// TIA Portal V17 program export: 17 tag tables, 178 data types, 56 data blocks, 100 code blocks (in call order from the OBs), 30 instance data blocks

VAR_GLOBAL   // PLC tag table "Default tag table"
   TIMER_PF_FEEDER_1_UNIT_01_LINE_1 AT %T21 : Timer;
   TIMER_PF_FEEDER_1_UNIT_01_LINE_2 AT %T22 : Timer;
   TIMER_PF_FEEDER_1_UNIT_02_LINE_1 AT %T23 : Timer;
   TIMER_PF_FEEDER_1_UNIT_02_LINE_2 AT %T24 : Timer;
   "Clock_Byte(1)" AT %MB0 : Byte;
   OK_DEL_NCU AT %M710.0 : Bool;
   Tag_1 AT %M45.0 : Bool;
   Tag_2 AT %M250.0 : Bool;
   Tag_3 AT %M71.0 : Bool;
   Tag_4 AT %M71.1 : Bool;
   Tag_5 AT %M71.2 : Bool;
   Tag_6 AT %M71.3 : Bool;
   Tag_7 AT %M71.4 : Bool;
   U01_OERLIKON_1_LINE_1_MEDICOAT_TIMER AT %T39 : Timer;   // UNIT 01 OERLIKON 1 LINE 1 MEDICOAT TIMER
   U01_OERLIKON_1_LINE_2_MEDICOAT_TIMER AT %T40 : Timer;   // UNIT 01 OERLIKON 1 LINE 2 MEDICOAT TIMER
   U02_OERLIKON_1_LINE_1_MEDICOAT_TIMER AT %T41 : Timer;   // UNIT 02 OERLIKON 1 LINE 1 MEDICOAT TIMER
   U02_OERLIKON_1_LINE_2_MEDICOAT_TIMER AT %T42 : Timer;   // UNIT 02 OERLIKON 1 LINE 2 MEDICOAT TIMER
   U01_COMBINER_MEDICOAT_TIMER AT %T44 : Timer;   // UNIT 01 COMBINER MEDICOAT TIMER
   U02_COMBINER_MEDICOAT_TIMER AT %T45 : Timer;   // UNIT 02 COMBINER MEDICOAT TIMER
   U01_LASER_HEAD_MEDICOAT_TIMER AT %T46 : Timer;   // UNIT 01 LASER HEAD MEDICOAT TIMER
   U02_LASER_HEAD_MEDICOAT_TIMER AT %T47 : Timer;   // UNIT 02 LASER HEAD MEDICOAT TIMER
   UNIT_01_PF1_L2_PRESS AT %MD26 : Real;
   UNIT_01_PF1_L1_PRESS AT %MD30 : Real;
   UNIT_01_PF2_L1_PRESS AT %MD34 : Real;
   U02_OERLIKON_2_LINE_2_MEDICOAT_TIMER AT %T43 : Timer;   // UNIT 02 OERLIKON 2 LINE 1 MEDICOAT TIMER
   TIMER_PF_FEEDER_2_UNIT_02_LINE_2 AT %T25 : Timer;
   Tag_8 AT %M445.4 : Bool;
   Tag_9 AT %T26 : Timer;
   Tag_10 AT %IW1810 : Int;
   COUNT_ANDER AT %MW448 : Int;
   PB_HOPPERS_MANUAL_MODE_SELECTED_LIGHT_Q AT %Q141.4 : Bool;   // MANUAL MODE SELECTED LIGHT OUTPUT
END_VAR

VAR_GLOBAL   // PLC tag table "TAGS_MARKS"
   Clock_Byte AT %MB1 : Byte;
   "M_0.1_SEC_10HZ" AT %M1.0 : Bool;   // 10HZ 0.1SEC
   "M_0.2_SEC_5Hz" AT %M1.1 : Bool;   // 5HZ 0.2SEC
   "M_0.4_SEC_2.5HZ" AT %M1.2 : Bool;   // 2.5HZ 0.4SEC
   "M_0.5_SEC_2HZ" AT %M1.3 : Bool;   // 2HZ 0.5SEC
   "M_0.8_SEC_1.25HZ" AT %M1.4 : Bool;   // 2.25HZ 0.8SEC
   "M_1.6_SEC_625HZ" AT %M1.6 : Bool;   // 0.625HZ 1.6SEC
   M_1_SEC_1HZ AT %M1.5 : Bool;   // 1HZ 1.0SEC
   "M_2_SEC_0.5HZ" AT %M1.7 : Bool;   // 0.5HZ 2.0SEC
   M_DUMMY_OFF AT %M0.3 : Bool;   // DUMMY OFF
   M_DUMMY_ON AT %M0.2 : Bool;   // DUMMY ON
   M_DUMMY_OUT AT %M0.4 : Bool;   // DUMMY OUT
   M_FIRST_SCAN AT %M0.6 : Bool;   // M FIRST SCAN
   M_NEW_START AT %M0.5 : Bool;   // NEW START / M NEW START
   M_ONE AT %M0.1 : Bool;   // ALWAYS ON
   M_REVISAR_FALTA_ALGO AT %M2.3 : Bool;   // REVISAR FALTA ALGO DE PROGRAMACIÓN
   M_TEMPORARY_USE_OEM AT %M5.0 : Bool;   // M_TEMPORARY_USE_OEM(CONFIGURE CORRECTLY AND DELETE) / M FOR TEMPORARY USE (OEM)
   M_ZERO AT %M0.0 : Bool;   // ALWAYS OFF
   NETWORK_CHECK AT %M0.7 : Bool;   // ADAPT NETWORK LOGIC ACCORDING TO MACHINE STRUCTURE
   Softkey_Input_Byte AT %IB124 : Byte;
END_VAR

VAR_GLOBAL   // PLC tag table "TAGS_IO_MPP_ITC_IPC_HT10"
   HT10_INS AT %I0.0 : "HT10_INPUTS";   // HT10 INPUTS
   HT10_OUTS AT %Q0.0 : "HT10_OUTPUTS";   // HT10 OUTPUTS
   MPP_INS AT %I120.0 : "MPP_INPUTS";   // MPP INPUTS
   MPP_OUT AT %Q120.0 : "MPP_OUTPUTS";   // MPP OUTPUTS
   TOUCH_PANEL_INPUT_1 AT %IB138 : Byte;   // TOUCH PANEL INPUT BYTE 1
   TOUCH_PANEL_INPUT_2 AT %IB139 : Byte;   // TOUCH PANEL INPUT BYTE 2
END_VAR

VAR_GLOBAL   // PLC tag table "TEMPORAL_TAG_PANI"
   PART_PRESENT_SENSOR_UNIT_1 AT %MW5000 : Int;
   Delay_Z11_Start AT %T10 : Timer;
   Delay_Z21_Start AT %T20 : Timer;
   U01_STA4_BRUSH_WORN_ALARM AT %M100.0 : Bool;
   U01_STA4_BRUSH_WORN_INPUT AT %M100.1 : Bool;
   U01_STA4_BRUSH_CHANGE_ACK AT %M100.2 : Bool;
END_VAR

VAR_GLOBAL   // PLC tag table "TAGS_IO_GENERAL_CLADDING"
   "/////_CRM_/////" AT %M6060.0 : Bool;   // /////_CRM_/////
   "/////_ELECTRICAL_CABINET_/////" AT %M6100.0 : Bool;   // /////_ELECTRICAL_CABINET_/////
   "/////_LINE_CONTACTOR_/////" AT %M6200.0 : Bool;   // /////_LINE_CONTACTOR_/////
   "/////_MPP_AND_SIGNAL_TOWER_/////" AT %M141.0 : Bool;   // /////_MPP_AND_SIGNAL_TOWER_/////
   "/////_POWER_SUPPLY_/////" AT %M6080.0 : Bool;   // /////_POWER_SUPPLY_/////
   "/////_SAFETY_DOORS_/////" AT %M6180.0 : Bool;   // /////_SAFETY_DOORS_/////
   CIRCUIT_BREAKER_230VAC_TRIPPED AT %I140.1 : Bool;   // 230 VAC CIRCUIT BREAKER TRIPPED
   CIRCUIT_BREAKER_FC04_TRIPPED AT %I140.0 : Bool;   // FC04 CIRCUIT BREAKER TRIPPED. FAN.
   CIRCUIT_BREAKER_FC35_1_TRIPPED AT %I140.5 : Bool;   // FC35.1 CIRCUIT BREAKER TRIPPED
   CIRCUIT_BREAKER_FC35_2_TRIPPED AT %I140.6 : Bool;   // FC35.2 CIRCUIT BREAKER TRIPPED
   CIRCUIT_BREAKER_FC35_3_TRIPPED AT %I140.7 : Bool;   // FC35.3 CIRCUIT BREAKER TRIPPED
   CONTROL_ON_Q AT %Q140.0 : Bool;   // CONTROL ON OUTPUT
   MAIN_CIRCUIT_BREAKER_I AT %M580.1 : Bool;   // MAIN CABINET CIRCUIT BREAKER TRIPPED INPUT
   PB_AUTO_CYCLE_LIGHT_Q AT %Q141.1 : Bool;   // AUTOMATIC CYCLE LIGHT OUTPUT
   PB_AUTO_MODE_SELECTED_LIGHT_Q AT %Q141.2 : Bool;   // AUTOMATIC MODE SELECTED LIGHT OUTPUT
   PB_IMMEDIATE_STOP_I AT %I144.3 : Bool;   // IMMEDIATE STOP INPUT
   PB_MANUAL_MODE_SELECTED_LIGHT_Q AT %Q141.3 : Bool;   // MANUAL MODE SELECTED LIGHT OUTPUT
   PB_RESET_FAULTS_I AT %I144.6 : Bool;   // RESET FAULTS INPUT
   PB_START_CYCLE_I AT %I144.2 : Bool;   // START CYCLE INPUT
   PS_24V_NOT_READY_DEV_1_I AT %I142.2 : Bool;   // POWER SUPPLY 24V NOT READY DEVICE 1 INPUT
   PS_24V_NOT_READY_DEV_2_I AT %I142.3 : Bool;   // POWER SUPPLY 24V NOT READY DEVICE 2 INPUT
   SIGNAL_TWR_BLUE_LIGHT_Q AT %M141.1 : Bool;   // SIGNAL TOWER BLUE LIGHT OUTPUT
   SIGNAL_TWR_GREEN_LIGHT_Q AT %Q141.5 : Bool;   // SIGNAL TOWER GREEN LIGHT OUTPUT
   SIGNAL_TWR_HOOTER_Q AT %M141.3 : Bool;   // SIGNAL TOWER HOOTER LIGHT OUTPUT
   SIGNAL_TWR_RED_LIGHT_Q AT %Q141.7 : Bool;   // SIGNAL TOWER RED LIGHT OUTPUT
   SIGNAL_TWR_WHITE_LIGHT_Q AT %M141.2 : Bool;   // SIGNAL TOWER WHITE LIGHT OUTPUT
   SIGNAL_TWR_YELLOW_LIGHT_Q AT %Q141.6 : Bool;   // SIGNAL TOWER YELLOW LIGHT OUTPUT
   PB_HOPPERS_AUTO_MODE_SELECTED_LIGHT_Q AT %Q141.0 : Bool;   // AUTOMATIC MODE SELECTED LIGHT OUTPUT
   PB_FEEDERS_AUTOMATIC_MODE_SELECT_I AT %I144.0 : Bool;   // AUTOMATIC MODE SELECT INPUT
   PB_FEEDERS_MANUAL_MODE_SELECT_I AT %I144.1 : Bool;   // MANUAL MODE SELECT INPUT
   PB_HOPPERS_MANUAL_MODE_SELECT_I AT %I142.6 : Bool;   // MANUAL MODE SELECT INPUT
   PB_HOPPERS_AUTOMATIC_MODE_SELECT_I AT %I142.5 : Bool;   // AUTOMATIC MODE SELECT INPUT
END_VAR

VAR_GLOBAL   // PLC tag table "TAGS_IO_HOPPERS_CLADDING"
   "//////////_HOPPERS_POWDER_FLOW_SENSORS_//////////" AT %M580.0 : Bool;
   "//////////_HOPPERS_WEIGHT_CONTROL_SENSORS_//////////" AT %M596.0 : Bool;
   "/////_HOPPER_JACKET_TEMPERATURE_CONTROL_/////" AT %M150.0 : Bool;   // /////_HOPPER_JACKET_TEMPERATURE_CONTROL/////
   "/////_HOPPER_LEVEL_SENSORS_/////" AT %M70.0 : Bool;   // /////_HOPPER_LEVEL_SENSORS_/////
   "/////_HOPPER_PRESSURE_SENSORS/////" AT %M510.0 : Bool;   // /////_HOPPER_PRESSURE_SENSORS/////
   "/////_HOPPERS_PRESSURE_CONTROLS_/////" AT %M160.0 : Bool;
   "/////_HOPPERS_VALVES_/////" AT %M75.0 : Bool;   // /////_HOPPERS_VALVES_/////
   HPPR_1_MOTOR_ENABLE_1 AT %Q140.4 : Bool;   // HOPPER 1 MOTOR ENABLE SIGNAL 1
   HPPR_1_MOTOR_ENABLE_2 AT %Q140.5 : Bool;   // HOPPER 1 MOTOR ENABLE SIGNAL 2
   HPPR_2_MOTOR_ENABLE_1 AT %Q140.6 : Bool;   // HOPPER 2 MOTOR ENABLE SIGNAL 1
   HPPR_2_MOTOR_ENABLE_2 AT %Q140.7 : Bool;   // HOPPER 2 MOTOR ENABLE SIGNAL 2
   HPPR_3_MOTOR_ENABLE_1 AT %Q142.2 : Bool;   // HOPPER 3 MOTOR ENABLE SIGNAL 1
   HPPR_3_MOTOR_ENABLE_2 AT %Q142.3 : Bool;   // HOPPER 3 MOTOR ENABLE SIGNAL 2
   HPPR_4_MOTOR_ENABLE_1 AT %Q142.4 : Bool;   // HOPPER 4 MOTOR ENABLE SIGNAL 1
   HPPR_4_MOTOR_ENABLE_2 AT %Q142.5 : Bool;   // HOPPER 4 MOTOR ENABLE SIGNAL 2
   HPPR_5_MOTOR_ENABLE_1 AT %Q142.6 : Bool;   // HOPPER 5 MOTOR ENABLE SIGNAL 1
   HPPR_5_MOTOR_ENABLE_2 AT %Q142.7 : Bool;   // HOPPER 5 MOTOR ENABLE SIGNAL 2
   U01_HOPPER_1_HIGH_LEVEL_SENSOR_I AT %I70.1 : Bool;   // UNIT 01 HOPPER 1 HIGH LEVEL SENSOR INPUT
   U01_HOPPER_1_LOW_LEVEL_SENSOR_I AT %I70.0 : Bool;   // UNIT 01 HOPPER 1 LOW LEVEL SENSOR INPUT
   U01_HOPPER_1_LOWER_JACKET_TEMP_CONTROL_I AT %MW162 : Word;   // UNIT 01 HOPPER 1 LOWER JACKET TEMPERATURE CONTROL INPUT
   U01_HOPPER_1_LOWER_JACKET_TEMP_CONTROL_Q AT %MW166 : Word;   // UNIT 01 HOPPER 1 LOWER JACKET TEMPERATURE CONTROL OUTPUT
   U01_HOPPER_1_POWDER_FLOW_SENSOR_I AT %IW580 : Word;   // UNIT 01 HOPPER 1 POWDER FLOW SENSOR INPUT
   U01_HOPPER_1_PRESSURE_SENSOR_I AT %IW510 : Word;   // UNIT 01HOPPER 1 PRESSURE SENSOR INPUT
   U01_HOPPER_1_UPPER_JACKET_TEMP_CONTROL_I AT %MW150 : Word;   // UNIT 01 HOPPER 1 UPPER JACKET TEMPERATURE CONTROL INPUT
   U01_HOPPER_1_UPPER_JACKET_TEMP_CONTROL_Q AT %MW155 : Word;   // UNIT 01 HOPPER 1 UPPER JACKET TEMPERATURE CONTROL OUTPUT
   U01_HOPPER_1_WEIGHT_SENSOR_I AT %IW596 : Word;   // UNIT 01 HOPPER 1 WEIGHT SENSOR INPUT
   U01_HOPPER_2_HIGH_LEVEL_SENSOR_I AT %I70.3 : Bool;   // UNIT 01 HOPPER 2 HIGH LEVEL SENSOR INPUT
   U01_HOPPER_2_LOW_LEVEL_SENSOR_I AT %I70.2 : Bool;   // UNIT 01 HOPPER 2 LOW LEVEL SENSOR INPUT
   U01_HOPPER_2_LOWER_JACKET_TEMP_CONTROL_I AT %MW168 : Word;   // UNIT 01 HOPPER 2 LOWER JACKET TEMPERATURE CONTROL INPUT
   U01_HOPPER_2_LOWER_JACKET_TEMP_CONTROL_Q AT %MW172 : Word;   // UNIT 01 HOPPER 2 LOWER JACKET TEMPERATURE CONTROL OUTPUT
   U01_HOPPER_2_POWDER_FLOW_SENSOR_I AT %IW582 : Word;   // UNIT 01 HOPPER 2 POWDER FLOW SENSOR INPUT
   U01_HOPPER_2_PRESSURE_SENSOR_I AT %IW518 : Word;   // UNIT 01HOPPER 2 PRESSURE SENSOR INPUT
   U01_HOPPER_2_UPPER_JACKET_TEMP_CONTROL_I AT %MW151 : Word;   // UNIT 01 HOPPER 2 UPPER JACKET TEMPERATURE CONTROL INPUT
   U01_HOPPER_2_UPPER_JACKET_TEMP_CONTROL_Q AT %MW156 : Word;   // UNIT 01 HOPPER 2 UPPER JACKET TEMPERATURE CONTROL OUTPUT
   U01_HOPPER_2_WEIGHT_SENSOR_I AT %IW598 : Word;   // UNIT 01 HOPPER 2 WEIGHT SENSOR INPUT
   U01_HPPR_1_CLEANING_VALVE_Q AT %M73.5 : Bool;   // UNIT 01 HOPPER 1 CLEANING VALVE OUTPUT
   U01_HPPR_1_FEEDBACK_PRESSURE_CONTROL_I AT %IW160 : Int;   // UNIT 01 HOPPER 1 FEEDBACK PRESSURE CONTROL INPUT
   U01_HPPR_1_PRESSURE_CONTROL_Q AT %QW160 : Int;   // UNIT 01 HOPPER 1 PRESSURE CONTROL OUTPUT
   U01_HPPR_1_PRESSURIZE_GAS_VALVE_Q AT %Q70.0 : Bool;   // UNIT 01 HOPPER 1 PRESSURIZE GAS VALVE OUTPUT
   U01_HPPR_1_RELIEF_GAS_VALVE_Q AT %Q70.1 : Bool;   // UNIT 01 HOPPER 1 RELIEF GAS VALVE OUTPUT
   U01_HPPR_1_TRANSF_POWDER_VALVE_Q AT %M1500.0 : Bool;   // UNIT 01 HOPPER 1 TRANSFER POWDER VALVE OUTPUT
   U01_HPPR_2_CLEANING_VALVE_Q AT %M73.6 : Bool;   // UNIT 01 HOPPER 2 CLEANING VALVE OUTPUT
   U01_HPPR_2_FEEDBACK_PRESSURE_CONTROL_I AT %IW162 : Int;   // UNIT 01 HOPPER 2 FEEDBACK PRESSURE CONTROL INPUT
   U01_HPPR_2_PRESSURE_CONTROL_Q AT %QW162 : Int;   // UNIT 01 HOPPER 2 PRESSURE CONTROL OUTPUT
   U01_HPPR_2_PRESSURIZE_GAS_VALVE_Q AT %Q70.2 : Bool;   // UNIT 01 HOPPER 2 PRESSURIZE GAS VALVE OUTPUT
   U01_HPPR_2_RELIEF_GAS_VALVE_Q AT %Q70.3 : Bool;   // UNIT 01 HOPPER 2 RELIEF GAS VALVE OUTPUT
   U01_HPPR_2_TRANSF_POWDER_VALVE_Q AT %M1500.1 : Bool;   // UNIT 01 HOPPER 2 TRANSFER POWDER VALVE OUTPUT
   U02_HOPPER_1_HIGH_LEVEL_SENSOR_I AT %I70.5 : Bool;   // UNIT 02 HOPPER 1 HIGH LEVEL SENSOR INPUT
   U02_HOPPER_1_LOW_LEVEL_SENSOR_I AT %I70.4 : Bool;   // UNIT 02 HOPPER 1 LOW LEVEL SENSOR INPUT
   U02_HOPPER_1_LOWER_JACKET_TEMP_CONTROL_I AT %MW176 : Word;   // UNIT 02 HOPPER 1 LOWER JACKET TEMPERATURE CONTROL INPUT
   U02_HOPPER_1_LOWER_JACKET_TEMP_CONTROL_Q AT %MW178 : Word;   // UNIT 02 HOPPER 1 LOWER JACKET TEMPERATURE CONTROL OUTPUT
   U02_HOPPER_1_POWDER_FLOW_SENSOR_I AT %IW584 : Word;   // UNIT 02 HOPPER 1 POWDER FLOW SENSOR INPUT
   U02_HOPPER_1_PRESSURE_SENSOR_I AT %IW526 : Word;   // UNIT 02 HOPPER 1 PRESSURE SENSOR INPUT
   U02_HOPPER_1_UPPER_JACKET_TEMP_CONTROL_I AT %MW152 : Word;   // UNIT 02 HOPPER 1 UPPER JACKET TEMPERATURE CONTROL INPUT
   U02_HOPPER_1_UPPER_JACKET_TEMP_CONTROL_Q AT %MW157 : Word;   // UNIT 02 HOPPER 1 UPPER JACKET TEMPERATURE CONTROL OUTPUT
   U02_HOPPER_1_WEIGHT_SENSOR_I AT %IW600 : Word;   // UNIT 02 HOPPER 1 WEIGHT SENSOR INPUT
   U02_HOPPER_2_HIGH_LEVEL_SENSOR_I AT %I70.7 : Bool;   // UNIT 02 HOPPER 2 HIGH LEVEL SENSOR INPUT
   U02_HOPPER_2_LOW_LEVEL_SENSOR_I AT %I70.6 : Bool;   // UNIT 02 HOPPER 2 LOW LEVEL SENSOR INPUT
   U02_HOPPER_2_LOWER_JACKET_TEMP_CONTROL_I AT %MW164 : Word;   // UNIT 02 HOPPER 2 LOWER JACKET TEMPERATURE CONTROL INPUT
   U02_HOPPER_2_LOWER_JACKET_TEMP_CONTROL_Q AT %MW174 : Word;   // UNIT 02 HOPPER 2 LOWER JACKET TEMPERATURE CONTROL OUTPUT
   U02_HOPPER_2_POWDER_FLOW_SENSOR_I AT %IW588 : Word;   // UNIT 02 HOPPER 2 POWDER FLOW SENSOR INPUT
   U02_HOPPER_2_PRESSURE_SENSOR_I AT %IW534 : Word;   // UNIT 02 HOPPER 2 PRESSURE SENSOR INPUT
   U02_HOPPER_2_UPPER_JACKET_TEMP_CONTROL_I AT %MW153 : Word;   // UNIT 02 HOPPER 2 UPPER JACKET TEMPERATURE CONTROL INPUT
   U02_HOPPER_2_UPPER_JACKET_TEMP_CONTROL_Q AT %MW158 : Word;   // UNIT 02 HOPPER 2 UPPER JACKET TEMPERATURE CONTROL OUTPUT
   U02_HOPPER_2_WEIGHT_SENSOR_I AT %IW602 : Word;   // UNIT 02 HOPPER 2 WEIGHT SENSOR INPUT
   U02_HOPPER_3_HIGH_LEVEL_SENSOR_I AT %I71.1 : Bool;   // UNIT 02 HOPPER 3 HIGH LEVEL SENSOR INPUT
   U02_HOPPER_3_LOW_LEVEL_SENSOR_I AT %I71.0 : Bool;   // UNIT 02 HOPPER 3 LOW LEVEL SENSOR INPUT
   U02_HOPPER_3_LOWER_JACKET_TEMP_CONTROL_I AT %MW170 : Word;   // UNIT 02 HOPPER 3 LOWER JACKET TEMPERATURE CONTROL INPUT
   U02_HOPPER_3_LOWER_JACKET_TEMP_CONTROL_Q AT %MW180 : Word;   // UNIT 02 HOPPER 3 LOWER JACKET TEMPERATURE CONTROL OUTPUT
   U02_HOPPER_3_POWDER_FLOW_SENSOR_I AT %IW590 : Word;   // UNIT 02 HOPPER 3 POWDER FLOW SENSOR INPUT
   U02_HOPPER_3_PRESSURE_SENSOR_I AT %IW542 : Word;   // UNIT 02 HOPPER 3 PRESSURE SENSOR INPUT
   U02_HOPPER_3_UPPER_JACKET_TEMP_CONTROL_I AT %MW154 : Word;   // UNIT 02 HOPPER 3 UPPER JACKET TEMPERATURE CONTROL INPUT
   U02_HOPPER_3_UPPER_JACKET_TEMP_CONTROL_Q AT %MW159 : Word;   // UNIT 02 HOPPER 3 UPPER JACKET TEMPERATURE CONTROL OUTPUT
   U02_HOPPER_3_WEIGHT_SENSOR_I AT %IW586 : Word;   // UNIT 02 HOPPER 3 WEIGHT SENSOR INPUT
   U02_HPPR_1_CLEANING_VALVE_Q AT %M73.7 : Bool;   // UNIT 02 HOPPER 1 CLEANING VALVE OUTPUT
   U02_HPPR_1_FEEDBACK_PRESSURE_CONTROL_I AT %IW164 : Int;   // UNIT 02 HOPPER 1 FEEDBACK PRESSURE CONTROL INPUT
   U02_HPPR_1_PRESSURE_CONTROL_Q AT %QW164 : Int;   // UNIT 02 HOPPER 1 PRESSURE CONTROL OUTPUT
   U02_HPPR_1_PRESSURIZE_GAS_VALVE_Q AT %Q70.4 : Bool;   // UNIT 02 HOPPER 1 PRESSURIZE GAS VALVE OUTPUT
   U02_HPPR_1_RELIEF_GAS_VALVE_Q AT %Q70.5 : Bool;   // UNIT 02 HOPPER 1 RELIEF GAS VALVE OUTPUT
   U02_HPPR_1_TRANSF_POWDER_VALVE_Q AT %M1500.2 : Bool;   // UNIT 02 HOPPER 1 TRANSFER POWDER VALVE OUTPUT
   U02_HPPR_2_CLEANING_VALVE_Q AT %M74.0 : Bool;   // UNIT 02 HOPPER 2 CLEANING VALVE OUTPUT
   U02_HPPR_2_FEEDBACK_PRESSURE_CONTROL_I AT %IW166 : Int;   // UNIT 02 HOPPER 2 FEEDBACK PRESSURE CONTROL INPUT
   U02_HPPR_2_PRESSURE_CONTROL_Q AT %QW166 : Int;   // UNIT 02 HOPPER 2 PRESSURE CONTROL OUTPUT
   U02_HPPR_2_PRESSURIZE_GAS_VALVE_Q AT %Q70.6 : Bool;   // UNIT 02 HOPPER 2 PRESSURIZE GAS VALVE OUTPUT
   U02_HPPR_2_RELIEF_GAS_VALVE_Q AT %Q70.7 : Bool;   // UNIT 02 HOPPER 2 RELIEF GAS VALVE OUTPUT
   U02_HPPR_2_TRANSF_POWDER_VALVE_Q AT %M1500.3 : Bool;   // UNIT 02 HOPPER 2 TRANSFER POWDER VALVE OUTPUT
   U02_HPPR_3_CLEANING_VALVE_Q AT %M1500.5 : Bool;   // UNIT 02 HOPPER 3 CLEANING VALVE OUTPUT
   U02_HPPR_3_FEEDBACK_PRESSURE_CONTROL_I AT %IW168 : Int;   // UNIT 02 HOPPER 3 FEEDBACK PRESSURE CONTROL INPUT
   U02_HPPR_3_PRESSURE_CONTROL_Q AT %QW170 : Int;   // UNIT 02 HOPPER 3 PRESSURE CONTROL OUTPUT
   U02_HPPR_3_PRESSURIZE_GAS_VALVE_Q AT %Q71.0 : Bool;   // UNIT 02 HOPPER 3 PRESSURIZE GAS VALVE OUTPUT
   U02_HPPR_3_RELIEF_GAS_VALVE_Q AT %Q71.1 : Bool;   // UNIT 02 HOPPER 3 RELIEF GAS VALVE OUTPUT
   U02_HPPR_3_TRANSF_POWDER_VALVE_Q AT %M1500.4 : Bool;   // UNIT 02 HOPPER 3 TRANSFER POWDER VALVE OUTPUT
END_VAR

VAR_GLOBAL   // PLC tag table "TAGS_IO_POWDER_FEEDERS_CLADDING"
   "//////////PF_HOPPERS_PRESSURE_SENSORS//////////" AT %M810.0 : Bool;
   "//////////POWDER_FEEDER_WEIGHT_CONTROL//////////" AT %M712.0 : Bool;
   "//////////POWDER_FLOW_SENSORS//////////" AT %M700.0 : Bool;
   U01_PF_1_WEIGHT_SENSOR_I AT %IW712 : Word;   // UNIT 01 POWDER FEEDER 1 WEIGHT SENSOR INPUT
   U02_COMBINER_FLOW_SENSOR_I AT %IW1706 : Word;   // UNIT 02 COMBINER FLOW SENSOR INPUT
   U02_OERLIKON_2_LINE_2_MEDICOAT_FLOW_CONTROL AT %MW16 : UInt;   // UNIT 02 OERLIKON 2 LINE 2 MEDICOAT FLOW CONTROL
   U02_OERLIKON_1_LINE_1_MEDICOAT_FLOW_CONTROL AT %IW1700 : Int;   // UNIT 02 OERLIKON 1 LINE 1 MEDICOAT FLOW CONTROL
   U02_COMBINER_MEDICOAT_FLOW_CONTROL AT %IW1708 : Int;   // UNIT 02 COMBINER MEDICOAT FLOW CONTROL
   U02_OERLIKON_2_LINE_1_MEDICOAT_FLOW_CONTROL AT %IW1704 : Int;   // UNIT 02 OERLIKON 2 LINE 1 MEDICOAT FLOW CONTROL
   U01_OERLIKON_1_LINE_1_MEDICOAT_FLOW_CONTROL AT %IW700 : Int;   // UNIT 01 OERLIKON 1 LINE 1 MEDICOAT FLOW CONTROL
   U02_PF_1_HPPR_1_PRESSURE_SENSOR_I AT %IW1818 : Word;   // UNIT 02 POWDER FEEDER 1 HOPPER 1 PRESSURE SENSOR INPUT
   U01_PF_1_HPPR_1_FLOW_SENSOR_I AT %MW700 : Word;   // UNIT 01 POWDER FEEDER 1 HOPPER 1 FLOW SENSOR INPUT
   U02_PF_2_HPPR_1_FLOW_SENSOR_I AT %MW1704 : Word;   // UNIT 02 POWDER FEEDER 2 HOPPER 1 FLOW SENSOR INPUT
   U01_PF_1_HPPR_1_PRESSURE_SENSOR_I AT %IW810 : Word;   // UNIT 01 POWDER FEEDER 1 HOPPER 1 PRESSURE SENSOR INPUT
   U02_PF_1_WEIGHT_SENSOR_I AT %MW1712 : Word;   // UNIT 02 POWDER FEEDER 1 WEIGHT SENSOR INPUT
   U02_PF_2_HPPR_1_PRESSURE_SENSOR_I AT %IW1822 : Word;   // UNIT 02 POWDER FEEDER 2 HOPPER 1 PRESSURE SENSOR INPUT
   U02_LASER_HEAD_FLOW_SENSOR_I AT %MW1708 : Word;   // UNIT 02 LASER HEAD FLOW SENSOR INPUT
   U02_PF_1_HPPR_2_PRESSURE_SENSOR_I AT %IW1820 : Word;   // UNIT 02 POWDER FEEDER 1 HOPPER 2 PRESSURE SENSOR INPUT
   U01_PF_1_HPPR_2_PRESSURE_SENSOR_I AT %IW812 : Word;   // UNIT 01 POWDER FEEDER 1 HOPPER 2 PRESSURE SENSOR INPUT
   U02_OERLIKON_1_LINE_2_MEDICOAT_FLOW_CONTROL AT %IW1702 : Int;   // UNIT 02 OERLIKON 1 LINE 2 MEDICOAT FLOW CONTROL
   U01_LASER_HEAD_FLOW_SENSOR_I AT %MW706 : Word;   // UNIT 01 LASER HEAD FLOW SENSOR INPUT
   U02_PF_2_WEIGHT_SENSOR_I AT %MW1714 : Word;   // UNIT 02 POWDER FEEDER 2 WEIGHT SENSOR INPUT
   U01_COMBINER_MEDICOAT_FLOW_CONTROL AT %IW708 : Int;   // UNIT 01 COMBINER MEDICOAT FLOW CONTROL
   U02_LASER_HEAD_MEDICOAT_CONTROL AT %IW1710 : Int;   // UNIT 02 LASER HEAD MEDICOAT FLOW CONTROL
   U01_COMBINER_FLOW_SENSOR_I AT %MW704 : Word;   // UNIT 01 COMBINER FLOW SENSOR INPUT
   U02_PF_1_HPPR_2_FLOW_SENSOR_I AT %MW1702 : Word;   // UNIT 02 POWDER FEEDER 1 HOPPER 2 FLOW SENSOR INPUT
   U01_OERLIKON_1_LINE_2_MEDICOAT_FLOW_CONTROL AT %IW702 : Int;   // UNIT 01 OERLIKON 1 LINE 2 MEDICOAT FLOW CONTROL
   U01_PF_1_HPPR_2_FLOW_SENSOR_I AT %MW702 : Word;   // UNIT 01 POWDER FEEDER 1 HOPPER 2 FLOW SENSOR INPUT
   U02_PF_1_HPPR_1_FLOW_SENSOR_I AT %MW1700 : Word;   // UNIT 02 POWDER FEEDER 1 HOPPER 1 FLOW SENSOR INPUT
   U01_LASER_HEAD_MEDICOAT_CONTROL AT %IW710 : Int;   // UNIT 01 LASER HEAD MEDICOAT FLOW CONTROL
   U02_PF1_L2_STIRRER_CURRENT AT %IW1716 : Int;
   U02_PF1_L1_STIRRER_CURRENT AT %IW1712 : Int;
   U02_PF2_L1_DISK_CURRENT AT %IW1722 : Int;
   U02_PF1_L2_DISK_CURRENT AT %IW1718 : Int;
   U01_PF1_L2_DISK_CURRENT AT %IW722 : Int;
   U01_PF1_L1_DISK_CURRENT AT %IW718 : Int;
   U01_PF1_L2_STIRRER_CURRENT AT %IW720 : Int;
   U01_PF1_L1_STIRRER_CURRENT AT %IW716 : Int;
   U02_PF1_L1_DISK_CURRENT AT %IW1714 : Int;
   U02_PF2_L2_STIRRER_CURRENT AT %IW1720 : Int;
END_VAR

VAR_GLOBAL   // PLC tag table "TAGS_IO_SERVICES_CLADDING"
   "/////_COOLING_CHILLER_/////" AT %M8305.6 : Bool;   // /////_COOLING_CHILLER_/////
   "/////_OTHER_CIRCUIT_BREAKERS_/////" AT %M8308.0 : Bool;   // /////_OTHER_CIRCUIT_BREAKERS_/////
   "/////_OTHER_CONTACTOR_/////" AT %M8309.5 : Bool;   // /////_OTHER_CONTACTOR_/////
END_VAR

VAR_GLOBAL   // PLC tag table "TAGS_IO_STIRRERS_CLADDING"
   "//////////_STIRRER_UNIT_01_HOPPER_1_//////////" AT %M500.0 : Bool;
   "//////////_STIRRER_UNIT_01_HOPPER_2_//////////" AT %M600.0 : Bool;
   "//////////_STIRRER_UNIT_02_HOPPER_1_//////////" AT %M2000.0 : Bool;
   "//////////_STIRRER_UNIT_02_HOPPER_2_//////////" AT %M800.0 : Bool;
   "//////////_STIRRER_UNIT_02_HOPPER_3_//////////" AT %M900.0 : Bool;
   U01_HPPR_1_STRR_ACTUAL_PHASE_CURRENT_FILTERED_INPUT AT %ID3016 : DInt;   // UNIT 01 HOPPER 1 STIRRER ACTUAL PHASE CURRENT FILTERED INPUT
   U01_HPPR_1_STRR_ACTUAL_PHASE_CURRENT_INPUT AT %ID3012 : DInt;   // UNIT 01 HOPPER 1 STIRRER ACTUAL PHASE CURRENT INPUT
   U01_HPPR_1_STRR_ACTUAL_POSITION_INPUT AT %ID3008 : DInt;   // UNIT 01 HOPPER 1 STIRRER STIRRER ACTUAL POSITON INPUT
   U01_HPPR_1_STRR_ACTUAL_TEMP_COM AT %IW3023 : Int;   // UNIT 01 HOPPER 1 STIRRER ACTUAL COM CARD TEMPERATURE
   U01_HPPR_1_STRR_ACTUAL_TEMP_POWER AT %IW3021 : Int;   // UNIT 01 HOPPER 1 STIRRER ACTUAL POWER STAGE TEMPERATURE
   U01_HPPR_1_STRR_ACTUAL_VELOCITY_INPUT AT %ID3004 : DInt;   // UNIT 01 HOPPER 1 STIRRER ACTUAL VELOCITY INPUT
   U01_HPPR_1_STRR_ENABLE_POWER_STAGE_OUTPUT AT %QB3005 : Byte;   // UNIT 01 HOPPER 1 STIRRER ENABLE POWER STAGE
   U01_HPPR_1_STRR_ERROR_CODE AT %IW3025 : Int;   // UNIT 01 HOPPER 1 STIRRER ERROR CODE
   U01_HPPR_1_STRR_IO_DIGITAL_OUTPUTS AT %QB3000 : Byte;   // UNIT 01 HOPPER 1 STIRRER IO DIGITAL OUTPUTS
   U01_HPPR_1_STRR_MODE_OF_OPERATION_OUTPUT AT %QB3006 : Byte;   // UNIT 01 HOPPER 1 STIRRER MODE OF OPERATION OUTPUT
   U01_HPPR_1_STRR_MOTOR_ENABLE_1_Q AT %M500.1 : Bool;   // UNIT 01 HOPPER 1 STIRRER MOTOR ENABLE 1 OUTPUT
   U01_HPPR_1_STRR_MOTOR_ENABLE_2_Q AT %M500.2 : Bool;   // UNIT 01 HOPPER 1 STIRRER MOTOR ENABLE 2 OUTPUT
   U01_HPPR_1_STRR_MOTOR_OUT_1 AT %Q3000.1 : Bool;   // UNIT 01 HOPPER 1 STIRRER MOTOR OUT 1
   U01_HPPR_1_STRR_MOTOR_OUT_2 AT %Q3000.2 : Bool;   // UNIT 01 HOPPER 1 STIRRER MOTOR OUT 2
   U01_HPPR_1_STRR_MOTOR_OUT_3 AT %Q3000.3 : Bool;   // UNIT 01 HOPPER 1 STIRRER MOTOR OUT 3
   U01_HPPR_1_STRR_MOTOR_STATUS_ENABLE AT %I3020.0 : Bool;   // UNIT 01 HOPPER 1 STIRRER MOTOR STATUS ENABLED
   U01_HPPR_1_STRR_MOTOR_STATUS_ENABLE_INPUT AT %I3000.0 : Bool;   // UNIT 01 HOPPER 1 STIRRER MOTOR STATUS ENABLE INPUT
   U01_HPPR_1_STRR_MOTOR_STATUS_ERROR AT %I3020.1 : Bool;   // UNIT 01 HOPPER 1 STIRRER MOTOR STATUS ERROR
   U01_HPPR_1_STRR_MOTOR_STATUS_ERROR_INPUT AT %I3000.1 : Bool;   // UNIT 01 HOPPER 1 STIRRER MOTOR STATUS ERROR INPUT
   U01_HPPR_1_STRR_MOTOR_STATUS_REACHED AT %I3020.4 : Bool;   // UNIT 01 HOPPER 1 STIRRER MOTOR STATUS REACHED
   U01_HPPR_1_STRR_MOTOR_STATUS_REACHED_INPUT AT %I3000.4 : Bool;   // UNIT 01 HOPPER 1 STIRRER MOTOR STATUS REACHED INPUT
   U01_HPPR_1_STRR_POWER_STAGE_HW_ENABLE_INPUTS AT %IB3020 : Byte;   // UNIT 01 HOPPER 1 STIRRER POWER STAGE STAGE HW ENABLE INPUTS
   U01_HPPR_1_STRR_STATUS_REGISTER_INPUTS AT %ID3000 : DInt;   // UNIT 01 HOPPER 1 STIRRER STATUS REGISTER INPUTS
   U01_HPPR_2_STRR_ACTUAL_PHASE_CURRENT_FILTERED_INPUT AT %ID3116 : DInt;   // UNIT 01 HOPPER 2 STIRRER ACTUAL PHASE CURRENT FILTERED INPUT
   U01_HPPR_2_STRR_ACTUAL_PHASE_CURRENT_INPUT AT %ID3112 : DInt;   // UNIT 01 HOPPER 2 STIRRER ACTUAL PHASE CURRENT INPUT
   U01_HPPR_2_STRR_ACTUAL_POSITION_INPUT AT %ID3108 : DInt;   // UNIT 01 HOPPER 2 STIRRER STIRRER ACTUAL POSITON INPUT
   U01_HPPR_2_STRR_ACTUAL_TEMP_COM AT %IW3123 : Int;   // UNIT 01 HOPPER 2 STIRRER ACTUAL COM CARD TEMPERATURE
   U01_HPPR_2_STRR_ACTUAL_TEMP_POWER AT %IW3121 : Int;   // UNIT 01 HOPPER 2 STIRRER ACTUAL POWER STAGE TEMPERATURE
   U01_HPPR_2_STRR_ACTUAL_VELOCITY_INPUT AT %ID3104 : DInt;   // UNIT 01 HOPPER 2 STIRRER ACTUAL VELOCITY INPUT
   U01_HPPR_2_STRR_ENABLE_POWER_STAGE_OUTPUT AT %QB3105 : Byte;   // UNIT 01 HOPPER 2 STIRRER ENABLE POWER STAGE
   U01_HPPR_2_STRR_ERROR_CODE AT %IW3125 : Int;   // UNIT 01 HOPPER 2 STIRRER ERROR CODE
   U01_HPPR_2_STRR_IO_DIGITAL_OUTPUTS AT %QB3100 : Byte;   // UNIT 01 HOPPER 2 STIRRER IO DIGITAL OUTPUTS
   U01_HPPR_2_STRR_MODE_OF_OPERATION_OUTPUT AT %QB3106 : Byte;   // UNIT 01 HOPPER 2 STIRRER MODE OF OPERATION OUTPUT
   U01_HPPR_2_STRR_MOTOR_ENABLE_1_Q AT %M600.1 : Bool;   // UNIT 01 HOPPER 2 STIRRER MOTOR ENABLE 1 OUTPUT
   U01_HPPR_2_STRR_MOTOR_ENABLE_2_Q AT %M600.2 : Bool;   // UNIT 01 HOPPER 2 STIRRER MOTOR ENABLE 2 OUTPUT
   U01_HPPR_2_STRR_MOTOR_OUT_1 AT %Q3100.1 : Bool;   // UNIT 01 HOPPER 2 STIRRER MOTOR OUT 1
   U01_HPPR_2_STRR_MOTOR_OUT_2 AT %Q3100.2 : Bool;   // UNIT 01 HOPPER 2 STIRRER MOTOR OUT 2
   U01_HPPR_2_STRR_MOTOR_OUT_3 AT %Q3100.3 : Bool;   // UNIT 01 HOPPER 2 STIRRER MOTOR OUT 3
   U01_HPPR_2_STRR_MOTOR_STATUS_ENABLE AT %I3120.0 : Bool;   // UNIT 01 HOPPER 2 STIRRER MOTOR STATUS ENABLED
   U01_HPPR_2_STRR_MOTOR_STATUS_ENABLE_INPUT AT %I3100.0 : Bool;   // UNIT 01 HOPPER 2 STIRRER MOTOR STATUS ENABLE INPUT
   U01_HPPR_2_STRR_MOTOR_STATUS_ERROR AT %I3120.1 : Bool;   // UNIT 01 HOPPER 2 STIRRER MOTOR STATUS ERROR
   U01_HPPR_2_STRR_MOTOR_STATUS_ERROR_INPUT AT %I3100.1 : Bool;   // UNIT 01 HOPPER 2 STIRRER MOTOR STATUS ERROR INPUT
   U01_HPPR_2_STRR_MOTOR_STATUS_REACHED AT %I3120.4 : Bool;   // UNIT 01 HOPPER 2 STIRRER MOTOR STATUS REACHED
   U01_HPPR_2_STRR_MOTOR_STATUS_REACHED_INPUT AT %I3100.4 : Bool;   // UNIT 01 HOPPER 2 STIRRER MOTOR STATUS REACHED INPUT
   U01_HPPR_2_STRR_POWER_STAGE_HW_ENABLE_INPUTS AT %IB3120 : Byte;   // UNIT 01 HOPPER 2 STIRRER POWER STAGE STAGE HW ENABLE INPUTS
   U01_HPPR_2_STRR_STATUS_REGISTER_INPUTS AT %ID3100 : DInt;   // UNIT 01 HOPPER 2 STIRRER STATUS REGISTER INPUTS
   U01_HPPR_2_STRR_VEL_TARGET_VALUE_OUTPUT AT %QD3101 : DInt;   // UNIT 01 HOPPER 2 STIRRER VELOCITY TARGET VALUE OUTPUT
   U01_HPPR1_STRR_VEL_TARGET_VALUE_OUTPUT AT %QD3001 : DInt;   // UNIT 01 HOPPER 1 STIRRER VELOCITY TARGET VALUE OUTPUT
   U02_HPPR_1_STRR_ACTUAL_PHASE_CURRENT_FILTERED_INPUT AT %ID3216 : DInt;   // UNIT 02 HOPPER 1 STIRRER ACTUAL PHASE CURRENT FILTERED INPUT
   U02_HPPR_1_STRR_ACTUAL_PHASE_CURRENT_INPUT AT %ID3212 : DInt;   // UNIT 02 HOPPER 1 STIRRER ACTUAL PHASE CURRENT INPUT
   U02_HPPR_1_STRR_ACTUAL_POSITION_INPUT AT %ID3208 : DInt;   // UNIT 02 HOPPER 1 STIRRER STIRRER ACTUAL POSITON INPUT
   U02_HPPR_1_STRR_ACTUAL_TEMP_COM AT %IW3223 : Int;   // UNIT 02 HOPPER 1 STIRRER ACTUAL COM CARD TEMPERATURE
   U02_HPPR_1_STRR_ACTUAL_TEMP_POWER AT %IW3221 : Int;   // UNIT 02 HOPPER 1 STIRRER ACTUAL POWER STAGE TEMPERATURE
   U02_HPPR_1_STRR_ACTUAL_VELOCITY_INPUT AT %ID3204 : DInt;   // UNIT 02 HOPPER 1 STIRRER ACTUAL VELOCITY INPUT
   U02_HPPR_1_STRR_ENABLE_POWER_STAGE_OUTPUT AT %QB3205 : Byte;   // UNIT 02 HOPPER 1 STIRRER ENABLE POWER STAGE
   U02_HPPR_1_STRR_ERROR_CODE AT %IW3225 : Int;   // UNIT 02 HOPPER 1 STIRRER ERROR CODE
   U02_HPPR_1_STRR_IO_DIGITAL_OUTPUTS AT %QB3200 : Byte;   // UNIT 02 HOPPER 1 STIRRER IO DIGITAL OUTPUTS
   U02_HPPR_1_STRR_MODE_OF_OPERATION_OUTPUT AT %QB3206 : Byte;   // UNIT 02 HOPPER 1 STIRRER MODE OF OPERATION OUTPUT
   U02_HPPR_1_STRR_MOTOR_ENABLE_1_Q AT %M700.1 : Bool;   // UNIT 02 HOPPER 1 STIRRER MOTOR ENABLE 1 OUTPUT
   U02_HPPR_1_STRR_MOTOR_ENABLE_2_Q AT %M700.2 : Bool;   // UNIT 02 HOPPER 1 STIRRER MOTOR ENABLE 2 OUTPUT
   U02_HPPR_1_STRR_MOTOR_OUT_1 AT %Q3200.1 : Bool;   // UNIT 02 HOPPER 1 STIRRER MOTOR OUT 1
   U02_HPPR_1_STRR_MOTOR_OUT_2 AT %Q3200.2 : Bool;   // UNIT 02 HOPPER 1 STIRRER MOTOR OUT 2
   U02_HPPR_1_STRR_MOTOR_OUT_3 AT %Q3200.3 : Bool;   // UNIT 02 HOPPER 1 STIRRER MOTOR OUT 3
   U02_HPPR_1_STRR_MOTOR_STATUS_ENABLE AT %I3220.0 : Bool;   // UNIT 02 HOPPER 1 STIRRER MOTOR STATUS ENABLED
   U02_HPPR_1_STRR_MOTOR_STATUS_ENABLE_INPUT AT %I3200.0 : Bool;   // UNIT 02 HOPPER 1 STIRRER MOTOR STATUS ENABLE INPUT
   U02_HPPR_1_STRR_MOTOR_STATUS_ERROR AT %I3220.1 : Bool;   // UNIT 02 HOPPER 1 STIRRER MOTOR STATUS ERROR
   U02_HPPR_1_STRR_MOTOR_STATUS_ERROR_INPUT AT %I3200.1 : Bool;   // UNIT 02 HOPPER 1 STIRRER MOTOR STATUS ERROR INPUT
   U02_HPPR_1_STRR_MOTOR_STATUS_REACHED AT %I3220.4 : Bool;   // UNIT 02 HOPPER 1 STIRRER MOTOR STATUS REACHED
   U02_HPPR_1_STRR_MOTOR_STATUS_REACHED_INPUT AT %I3200.4 : Bool;   // UNIT 02 HOPPER 1 STIRRER MOTOR STATUS REACHED INPUT
   U02_HPPR_1_STRR_POWER_STAGE_HW_ENABLE_INPUTS AT %IB3220 : Byte;   // UNIT 02 HOPPER 1 STIRRER POWER STAGE STAGE HW ENABLE INPUTS
   U02_HPPR_1_STRR_STATUS_REGISTER_INPUTS AT %ID3200 : DInt;   // UNIT 02 HOPPER 1 STIRRER STATUS REGISTER INPUTS
   U02_HPPR_1_STRR_VEL_TARGET_VALUE_OUTPUT AT %QD3201 : DInt;   // UNIT 02 HOPPER 1 STIRRER VELOCITY TARGET VALUE OUTPUT
   U02_HPPR_2_STRR_ACTUAL_PHASE_CURRENT_FILTERED_INPUT AT %ID3316 : DInt;   // UNIT 02 HOPPER 2 STIRRER ACTUAL PHASE CURRENT FILTERED INPUT
   U02_HPPR_2_STRR_ACTUAL_PHASE_CURRENT_INPUT AT %ID3312 : DInt;   // UNIT 02 HOPPER 2 STIRRER ACTUAL PHASE CURRENT INPUT
   U02_HPPR_2_STRR_ACTUAL_POSITION_INPUT AT %ID3308 : DInt;   // UNIT 02 HOPPER 2 STIRRER STIRRER ACTUAL POSITON INPUT
   U02_HPPR_2_STRR_ACTUAL_TEMP_COM AT %IW3323 : Int;   // UNIT 02 HOPPER 2 STIRRER ACTUAL COM CARD TEMPERATURE
   U02_HPPR_2_STRR_ACTUAL_TEMP_POWER AT %IW3321 : Int;   // UNIT 02 HOPPER 2 STIRRER ACTUAL POWER STAGE TEMPERATURE
   U02_HPPR_2_STRR_ACTUAL_VELOCITY_INPUT AT %ID3304 : DInt;   // UNIT 02 HOPPER 2 STIRRER ACTUAL VELOCITY INPUT
   U02_HPPR_2_STRR_ENABLE_POWER_STAGE_OUTPUT AT %QB3305 : Byte;   // UNIT 02 HOPPER 2 STIRRER ENABLE POWER STAGE
   U02_HPPR_2_STRR_ERROR_CODE AT %IW3325 : Int;   // UNIT 02 HOPPER 2 STIRRER ERROR CODE
   U02_HPPR_2_STRR_IO_DIGITAL_OUTPUTS AT %QB3300 : Byte;   // UNIT 02 HOPPER 2 STIRRER IO DIGITAL OUTPUTS
   U02_HPPR_2_STRR_MODE_OF_OPERATION_OUTPUT AT %QB3306 : Byte;   // UNIT 02 HOPPER 2 STIRRER MODE OF OPERATION OUTPUT
   U02_HPPR_2_STRR_MOTOR_ENABLE_1_Q AT %M800.1 : Bool;   // UNIT 02 HOPPER 2 STIRRER MOTOR ENABLE 1 OUTPUT
   U02_HPPR_2_STRR_MOTOR_ENABLE_2_Q AT %M800.2 : Bool;   // UNIT 02 HOPPER 2 STIRRER MOTOR ENABLE 2 OUTPUT
   U02_HPPR_2_STRR_MOTOR_OUT_1 AT %Q3300.1 : Bool;   // UNIT 02 HOPPER 2 STIRRER MOTOR OUT 1
   U02_HPPR_2_STRR_MOTOR_OUT_2 AT %Q3300.2 : Bool;   // UNIT 02 HOPPER 2 STIRRER MOTOR OUT 2
   U02_HPPR_2_STRR_MOTOR_OUT_3 AT %Q3300.3 : Bool;   // UNIT 02 HOPPER 2 STIRRER MOTOR OUT 3
   U02_HPPR_2_STRR_MOTOR_STATUS_ENABLE AT %I3320.0 : Bool;   // UNIT 02 HOPPER 2 STIRRER MOTOR STATUS ENABLED
   U02_HPPR_2_STRR_MOTOR_STATUS_ENABLE_INPUT AT %I3300.0 : Bool;   // UNIT 02 HOPPER 2 STIRRER MOTOR STATUS ENABLE INPUT
   U02_HPPR_2_STRR_MOTOR_STATUS_ERROR AT %I3320.1 : Bool;   // UNIT 02 HOPPER 2 STIRRER MOTOR STATUS ERROR
   U02_HPPR_2_STRR_MOTOR_STATUS_ERROR_INPUT AT %I3300.1 : Bool;   // UNIT 02 HOPPER 2 STIRRER MOTOR STATUS ERROR INPUT
   U02_HPPR_2_STRR_MOTOR_STATUS_REACHED AT %I3320.4 : Bool;   // UNIT 02 HOPPER 2 STIRRER MOTOR STATUS REACHED
   U02_HPPR_2_STRR_MOTOR_STATUS_REACHED_INPUT AT %I3300.4 : Bool;   // UNIT 02 HOPPER 2 STIRRER MOTOR STATUS REACHED INPUT
   U02_HPPR_2_STRR_POWER_STAGE_HW_ENABLE_INPUTS AT %IB3320 : Byte;   // UNIT 02 HOPPER 2 STIRRER POWER STAGE STAGE HW ENABLE INPUTS
   U02_HPPR_2_STRR_STATUS_REGISTER_INPUTS AT %ID3300 : DInt;   // UNIT 02 HOPPER 2 STIRRER STATUS REGISTER INPUTS
   U02_HPPR_2_STRR_VEL_TARGET_VALUE_OUTPUT AT %QD3301 : DInt;   // UNIT 02 HOPPER 2 STIRRER VELOCITY TARGET VALUE OUTPUT
   U02_HPPR_3_STRR_ACTUAL_PHASE_CURRENT_FILTERED_INPUT AT %ID3416 : DInt;   // UNIT 02 HOPPER 3 STIRRER ACTUAL PHASE CURRENT FILTERED INPUT
   U02_HPPR_3_STRR_ACTUAL_PHASE_CURRENT_INPUT AT %ID3412 : DInt;   // UNIT 02 HOPPER 3 STIRRER ACTUAL PHASE CURRENT INPUT
   U02_HPPR_3_STRR_ACTUAL_POSITION_INPUT AT %ID3408 : DInt;   // UNIT 02 HOPPER 3 STIRRER STIRRER ACTUAL POSITON INPUT
   U02_HPPR_3_STRR_ACTUAL_TEMP_COM AT %IW3423 : Int;   // UNIT 02 HOPPER 3 STIRRER ACTUAL COM CARD TEMPERATURE
   U02_HPPR_3_STRR_ACTUAL_TEMP_POWER AT %IW3421 : Int;   // UNIT 02 HOPPER 3 STIRRER ACTUAL POWER STAGE TEMPERATURE
   U02_HPPR_3_STRR_ACTUAL_VELOCITY_INPUT AT %ID3404 : DInt;   // UNIT 02 HOPPER 3 STIRRER ACTUAL VELOCITY INPUT
   U02_HPPR_3_STRR_ENABLE_POWER_STAGE_OUTPUT AT %QB3405 : Byte;   // UNIT 02 HOPPER 3 STIRRER ENABLE POWER STAGE
   U02_HPPR_3_STRR_ERROR_CODE AT %IW3425 : Int;   // UNIT 02 HOPPER 3 STIRRER ERROR CODE
   U02_HPPR_3_STRR_IO_DIGITAL_OUTPUTS AT %QB3400 : Byte;   // UNIT 02 HOPPER 3 STIRRER IO DIGITAL OUTPUTS
   U02_HPPR_3_STRR_MODE_OF_OPERATION_OUTPUT AT %QB3406 : Byte;   // UNIT 02 HOPPER 3 STIRRER MODE OF OPERATION OUTPUT
   U02_HPPR_3_STRR_MOTOR_ENABLE_1_Q AT %M900.1 : Bool;   // UNIT 02 HOPPER 3 STIRRER MOTOR ENABLE 1 OUTPUT
   U02_HPPR_3_STRR_MOTOR_ENABLE_2_Q AT %M900.2 : Bool;   // UNIT 02 HOPPER 3 STIRRER MOTOR ENABLE 2 OUTPUT
   U02_HPPR_3_STRR_MOTOR_OUT_1 AT %Q3400.1 : Bool;   // UNIT 02 HOPPER 3 STIRRER MOTOR OUT 1
   U02_HPPR_3_STRR_MOTOR_OUT_2 AT %Q3400.2 : Bool;   // UNIT 02 HOPPER 3 STIRRER MOTOR OUT 2
   U02_HPPR_3_STRR_MOTOR_OUT_3 AT %Q3400.3 : Bool;   // UNIT 02 HOPPER 3 STIRRER MOTOR OUT 3
   U02_HPPR_3_STRR_MOTOR_STATUS_ENABLE AT %I3420.0 : Bool;   // UNIT 02 HOPPER 3 STIRRER MOTOR STATUS ENABLED
   U02_HPPR_3_STRR_MOTOR_STATUS_ENABLE_INPUT AT %I3400.0 : Bool;   // UNIT 02 HOPPER 3 STIRRER MOTOR STATUS ENABLE INPUT
   U02_HPPR_3_STRR_MOTOR_STATUS_ERROR AT %I3420.1 : Bool;   // UNIT 02 HOPPER 3 STIRRER MOTOR STATUS ERROR
   U02_HPPR_3_STRR_MOTOR_STATUS_ERROR_INPUT AT %I3400.1 : Bool;   // UNIT 02 HOPPER 3 STIRRER MOTOR STATUS ERROR INPUT
   U02_HPPR_3_STRR_MOTOR_STATUS_REACHED AT %I3420.4 : Bool;   // UNIT 02 HOPPER 3 STIRRER MOTOR STATUS REACHED
   U02_HPPR_3_STRR_MOTOR_STATUS_REACHED_INPUT AT %I3400.4 : Bool;   // UNIT 02 HOPPER 3 STIRRER MOTOR STATUS REACHED INPUT
   U02_HPPR_3_STRR_POWER_STAGE_HW_ENABLE_INPUTS AT %IB3420 : Byte;   // UNIT 02 HOPPER 3 STIRRER POWER STAGE STAGE HW ENABLE INPUTS
   U02_HPPR_3_STRR_STATUS_REGISTER_INPUTS AT %ID3400 : DInt;   // UNIT 02 HOPPER 3 STIRRER STATUS REGISTER INPUTS
   U02_HPPR_3_STRR_VEL_TARGET_VALUE_OUTPUT AT %QD3401 : DInt;   // UNIT 02 HOPPER 3 STIRRER VELOCITY TARGET VALUE OUTPUT
END_VAR

VAR_GLOBAL   // PLC tag table "TAGS_SAFETY_IO_PROGRAM"
   FEEDBACK_OFF_E_STOP_IN AT %I143.1 : Bool;   // FEEDBACK OFF E-STOP INPUT
   FEEDBACK_OFF_E_STOP_RST_STR_IN AT %I143.2 : Bool;   // FEEDBACK OFF E-STOP RESET START INPUT
   FEEDBACK_OFF_MACHINE_E_STOP_IN AT %M10030.2 : Bool;   // FEEDBACK OFF MACHINE E-STOP INPUT
   FEEDBACK_OFF_MACHINE_E_STOP_RST_STR_IN AT %M10030.3 : Bool;   // FEEDBACK OFF MACHINE E-STOP RESET START INPUT
   SAFE_INPUT_MACH_E_STOP AT %I300.0 : Bool;   // SAFETY INPUT MACHINE EMERGENCY STOP
   SAFE_OUT_E_STOP_OK AT %Q330.0 : Bool;   // SAFETY OUTPUT EMERGENCY STOP OK
   SAFE_OUT_MACHINE_E_STOP_OK AT %M10050.1 : Bool;   // SAFETY OUTPUT EMERGENCY STOP OK
END_VAR

VAR_GLOBAL   // PLC tag table "TAGS_IO_CYLINDERS_CLADDING"
   "/////_SAFETY_BRAKES_/////" AT %M1200.0 : Bool;   // /////_SAFETY_BRAKES_/////
   SAFETY_BRAKE_AXIS_Z13_BLCKD_I AT %I570.5 : Bool;   // AXIS Z13 BRAKE BLOCKED INPUT
   SAFETY_BRAKE_AXIS_Z13_UNBLCKD_I AT %I570.6 : Bool;   // AXIS Z13 BRAKE UNBLOCKED INPUT
   SAFETY_BRAKE_AXIS_Z13_MAINT_BLCKD_I AT %M1200.3 : Bool;   // SAFETY BRAKE AXIS Z13 MAINTENANCE BRAKE BLOCKED INPUT
   SAFETY_BRAKE_AXIS_Z13_MAINT_UNBLCKD_I AT %M1200.4 : Bool;   // SAFETY BRAKE AXIS Z13 MAINTENANCE BRAKE UNBLOCKED INPUT
   SAFETY_BRAKE_AXIS_Z13_BLCK_Q AT %M1200.5 : Bool;   // SAFETY BRAKE AXIS Z13 BLOCK OUTPUT
   SAFETY_BRAKE_AXIS_Z23_BLCKD_I AT %I1570.5 : Bool;   // SAFETY BRAKE AXIS Z23 BLOCKED INPUT
   SAFETY_BRAKE_AXIS_Z23_UNBLCKD_I AT %I1570.6 : Bool;   // SAFETY BRAKE AXIS Z23 UNBLOCKED INPUT
   SAFETY_BRAKE_AXIS_Z23_MAINT_BLCKD_I AT %M1201.1 : Bool;   // SAFETY BRAKE AXIS Z23 MAINTENANCE BRAKE BLOCKED INPUT
   SAFETY_BRAKE_AXIS_Z23_MAINT_UNBLCKD_I AT %M1201.2 : Bool;   // SAFETY BRAKE AXIS Z23 MAINTENANCE BRAKE UNBLOCKED INPUT
   SAFETY_BRAKE_AXIS_Z23_BLCK_Q AT %M1201.3 : Bool;   // SAFETY BRAKE AXIS Z23 BLOCK OUTPUT
   "/////_UP_SEALING_U01_STRUCTURE_/////" AT %M1201.5 : Bool;   // /////_UP_SEALING_U01_STRUCTURE_/////
   UP_SEALING_U01_OPND_I_1 AT %I490.2 : Bool;   // UP SEALING UNIT 01 STRUCTURE OPENED INPUT 1
   UP_SEALING_U01_OPND_I_2 AT %I490.4 : Bool;   // UP SEALING UNIT 01 STRUCTURE OPENED INPUT 2
   UP_SEALING_U01_OPND_I_3 AT %I470.4 : Bool;   // UP SEALING UNIT 01 STRUCTURE OPENED INPUT 3
   UP_SEALING_U01_OPND_I_4 AT %I470.6 : Bool;   // UP SEALING UNIT 01 STRUCTURE OPENED INPUT 4
   UP_SEALING_U01_CLSD_I_1 AT %I490.3 : Bool;   // UP SEALING UNIT 01 STRUCTURE CLOSED INPUT 1
   UP_SEALING_U01_CLSD_I_2 AT %I490.5 : Bool;   // UP SEALING UNIT 01 STRUCTURE CLOSED INPUT 2
   UP_SEALING_U01_CLSD_I_3 AT %I470.5 : Bool;   // UP SEALING UNIT 01 STRUCTURE CLOSED INPUT 3
   UP_SEALING_U01_CLSD_I_4 AT %I470.7 : Bool;   // UP SEALING UNIT 01 STRUCTURE CLOSED INPUT 4
   "/////_DOWN_SEALING_U01_STRUCTURE_/////" AT %M1203.0 : Bool;   // /////_DOWN_SEALING_U01_STRUCTURE_/////
   DOWN_SEALING_U01_OPND_I_1 AT %M1203.1 : Bool;   // DOWN SEALING UNIT 01 STRUCTURE OPENED INPUT 1
   DOWN_SEALING_U01_OPND_I_2 AT %M1203.2 : Bool;   // DOWN SEALING UNIT 01 STRUCTURE OPENED INPUT 2
   DOWN_SEALING_U01_OPND_I_3 AT %I490.7 : Bool;   // DOWN SEALING UNIT 01 STRUCTURE OPENED INPUT 3
   DOWN_SEALING_U01_OPND_I_4 AT %I480.1 : Bool;   // DOWN SEALING UNIT 01 STRUCTURE OPENED INPUT 4
   DOWN_SEALING_U01_CLSD_I_1 AT %M1203.5 : Bool;   // DOWN SEALING UNIT 01 STRUCTURE CLOSED INPUT 1
   DOWN_SEALING_U01_CLSD_I_2 AT %M1203.6 : Bool;   // DOWN SEALING UNIT 01 STRUCTURE CLOSED INPUT 2
   DOWN_SEALING_U01_CLSD_I_3 AT %I490.6 : Bool;   // DOWN SEALING UNIT 01 STRUCTURE CLOSED INPUT 3
   DOWN_SEALING_U01_CLSD_I_4 AT %I480.0 : Bool;   // DOWN SEALING UNIT 01 STRUCTURE CLOSED INPUT 4
   "/////_UNIT_01_BEAM_SAMPLER/////" AT %M1207.1 : Bool;   // /////_UNIT_01_BEAM_SAMPLER/////
   U01_ST4_BEAM_SAMPLER_BLOW_I AT %M1207.2 : Bool;   // UNIT 01 BEAM SAMPLER BLOWING INPUT
   U01_ST4_BEAM_SAMPLER_PRESSURIZED_I AT %M1207.3 : Bool;   // UNIT 01 BEAM SAMPLER PRESSURIZED INPUT
   U01_ST4_BEAM_SAMPLER_BLOW_Q AT %M1207.4 : Bool;   // UNIT 01 BEAM SAMPLER BLOW OUTPUT STATION 4
   "/////_UNIT_01_DUST_EXTRACTION_1/////" AT %M1207.5 : Bool;   // /////_UNIT_01_DUST_EXTRACTION_1/////
   U01_DUST_EXTRAC_1_SWTCHD_ON_I AT %M1207.6 : Bool;   // UNIT 01 DUST EXTRACCION 1 SWITCHED ON INPUT (Flow Present)
   U01_DUST_EXTRAC_1_SWTCHD_OFF_I AT %M1207.7 : Bool;   // UNIT 01 DUST EXTRACCION 1 SWITCHED OFF INPUT
   U01_DUST_EXTRAC_1_SWTCH_OFF_Q AT %M1208.1 : Bool;   // UNIT 01 DUST EXTRACCION 1 SWITCH OFF OUTPUT
   "/////_UNIT_01_DUST_EXTRACTION_2/////" AT %M1208.2 : Bool;   // /////_UNIT_01_DUST_EXTRACTION_2/////
   U01_DUST_EXTRAC_2_SWTCHD_ON_I AT %M1208.3 : Bool;   // UNIT 01 DUST EXTRACCION 2 SWITCHED ON INPUT (Flow Present)
   U01_DUST_EXTRAC_2_SWTCHD_OFF_I AT %M1208.4 : Bool;   // UNIT 01 DUST EXTRACCION 2 SWITCHED OFF INPUT
   U01_DUST_EXTRAC_2_SWTCH_ON_Q AT %M1208.5 : Bool;   // UNIT 01 DUST EXTRACCION 2 SWITCH ON OUTPUT
   U01_DUST_EXTRAC_2_SWTCH_OFF_Q AT %M1208.6 : Bool;   // UNIT 01 DUST EXTRACCION 2 SWITCH OFF OUTPUT
   "/////_UNIT_01_DUST_EXTRACTION_3/////" AT %M1208.7 : Bool;   // /////_UNIT_01_DUST_EXTRACTION_3/////
   U01_DUST_EXTRAC_3_SWTCHD_ON_I AT %M1209.0 : Bool;   // UNIT 01 DUST EXTRACCION 3 SWITCHED ON INPUT (Flow Present)
   U01_DUST_EXTRAC_3_SWTCHD_OFF_I AT %M1209.1 : Bool;   // UNIT 01 DUST EXTRACCION 3 SWITCHED OFF INPUT
   U01_DUST_EXTRAC_3_SWTCH_OFF_Q AT %M1209.3 : Bool;   // UNIT 01 DUST EXTRACCION 3 SWITCH OFF OUTPUT
   "/////_UNIT_01_DUST_EXTRACTION_4/////" AT %M1209.4 : Bool;   // /////_UNIT_01_DUST_EXTRACTION_4/////
   U01_DUST_EXTRAC_4_SWTCHD_ON_I AT %M1209.5 : Bool;   // UNIT 01 DUST EXTRACCION 4 SWITCHED ON INPUT (Flow Present)
   U01_DUST_EXTRAC_4_SWTCHD_OFF_I AT %M1209.6 : Bool;   // UNIT 01 DUST EXTRACCION 4 SWITCHED OFF INPUT
   U01_DUST_EXTRAC_4_SWTCH_OFF_Q AT %M1210.0 : Bool;   // UNIT 01 DUST EXTRACCION 4 SWITCH OFF OUTPUT
   "/////_UNIT_01_ANGULAR_LOCATOR_/////" AT %M1210.6 : Bool;
   U01_ANGULAR_LOCATOR_LCTD_I AT %I578.0 : Bool;
   U01_ANGULAR_LOCATOR_RTND_I AT %I578.1 : Bool;
   "/////_UNIT_01_AXIAL_LOCATOR_/////" AT %M1211.3 : Bool;
   U01_AXIAL_LOCATOR_LCTD_I AT %I578.2 : Bool;
   U01_AXIAL_LOCATOR_RTND_I AT %I578.3 : Bool;
   "/////_UNIT_01_STATION_4_BRUSH/////" AT %M1212.0 : Bool;   // /////_UNIT_01_STATION_4_BRUSH/////
   U01_ST4_BRUSH_LCTD_I AT %M1212.1 : Bool;   // UNIT 01 STATION 4 BRUSH LOCATED INPUT
   U01_ST4_BRUSH_RTND_I AT %M1212.2 : Bool;   // UNIT 01 STATION 4 BRUSH RETURNED INPUT
   U01_ST4_BRUSH_LCT_Q AT %M1212.3 : Bool;
   U01_ST4_BRUSH_RTN_Q AT %M1212.4 : Bool;
   "/////_UP_SEALING_U02_STRUCTURE_/////" AT %M1212.5 : Bool;   // /////_UP_SEALING_U02_STRUCTURE_/////
   UP_SEALING_U02_OPND_I_1 AT %I1490.2 : Bool;   // UP SEALING UNIT 02 STRUCTURE OPENED INPUT 1
   UP_SEALING_U02_OPND_I_2 AT %I1490.4 : Bool;   // UP SEALING UNIT 02 STRUCTURE OPENED INPUT 2
   UP_SEALING_U02_OPND_I_3 AT %I1470.4 : Bool;   // UP SEALING UNIT 02 STRUCTURE OPENED INPUT 3
   UP_SEALING_U02_OPND_I_4 AT %I1470.6 : Bool;   // UP SEALING UNIT 02 STRUCTURE OPENED INPUT 4
   UP_SEALING_U02_CLSD_I_1 AT %I1490.3 : Bool;   // UP SEALING UNIT 02 STRUCTURE CLOSED INPUT 1
   UP_SEALING_U02_CLSD_I_2 AT %I1490.5 : Bool;   // UP SEALING UNIT 02 STRUCTURE CLOSED INPUT 2
   UP_SEALING_U02_CLSD_I_3 AT %I1470.5 : Bool;   // UP SEALING UNIT 02 STRUCTURE CLOSED INPUT 3
   UP_SEALING_U02_CLSD_I_4 AT %I1470.7 : Bool;   // UP SEALING UNIT 02 STRUCTURE CLOSED INPUT 4
   "/////_DOWN_SEALING_U02_STRUCTURE_/////" AT %M1214.0 : Bool;   // /////_DOWN_SEALING_U02_STRUCTURE_/////
   DOWN_SEALING_U02_OPND_I_1 AT %M1214.1 : Bool;   // DOWN SEALING UNIT 02 STRUCTURE OPENED INPUT 1
   DOWN_SEALING_U02_OPND_I_2 AT %M1214.2 : Bool;   // DOWN SEALING UNIT 02 STRUCTURE OPENED INPUT 2
   DOWN_SEALING_U02_OPND_I_3 AT %I1490.7 : Bool;   // DOWN SEALING UNIT 02 STRUCTURE OPENED INPUT 3
   DOWN_SEALING_U02_OPND_I_4 AT %I1480.1 : Bool;   // DOWN SEALING UNIT 02 STRUCTURE OPENED INPUT 4
   DOWN_SEALING_U02_CLSD_I_1 AT %M1214.5 : Bool;   // DOWN SEALING UNIT 02 STRUCTURE CLOSED INPUT 1
   DOWN_SEALING_U02_CLSD_I_2 AT %M1214.6 : Bool;   // DOWN SEALING UNIT 02 STRUCTURE CLOSED INPUT 2
   DOWN_SEALING_U02_CLSD_I_3 AT %I1490.6 : Bool;   // DOWN SEALING UNIT 02 STRUCTURE CLOSED INPUT 3
   DOWN_SEALING_U02_CLSD_I_4 AT %I1480.0 : Bool;   // DOWN SEALING UNIT 02 STRUCTURE CLOSED INPUT 4
   "/////_UNIT_02_BEAM_SAMPLER/////" AT %M1215.3 : Bool;   // /////_UNIT_02_BEAM_SAMPLER/////
   U02_ST4_BEAM_SAMPLER_BLOW_I AT %M1215.4 : Bool;   // UNIT 02 BEAM SAMPLER BLOWING INPUT
   U02_ST4_BEAM_SAMPLER_PRESSURIZED_I AT %M1215.5 : Bool;   // UNIT 02 BEAM SAMPLER PRESSURIZED INPUT
   U02_ST4_BEAM_SAMPLER_BLOW_Q AT %M1215.6 : Bool;   // UNIT 01 BEAM SAMPLER BLOW OUTPUT STATION 4
   "/////_UNIT_02_DUST_EXTRACTION_1_/////" AT %M1215.7 : Bool;   // /////_UNIT_02_DUST_EXTRACTION_1/////
   U02_DUST_EXTRAC_1_SWTCHD_ON_I AT %M1216.0 : Bool;   // UNIT 02 DUST EXTRACCION 1 SWITCHED ON INPUT (Flow Present)
   U02_DUST_EXTRAC_1_SWTCHD_OFF_I AT %M1216.1 : Bool;   // UNIT 02 DUST EXTRACCION 1 SWITCHED OFF INPUT
   U02_DUST_EXTRAC_1_SWTCH_OFF_Q AT %M1216.3 : Bool;   // UNIT 02 DUST EXTRACCION 1 SWITCH OFF OUTPUT
   "/////_UNIT_02_DUST_EXTRACTION_2_/////" AT %M1216.4 : Bool;   // /////_UNIT_02_DUST_EXTRACTION_2/////
   U02_DUST_EXTRAC_2_SWTCHD_ON_I AT %M1216.5 : Bool;   // UNIT 02 DUST EXTRACCION 2 SWITCHED ON INPUT (Flow Present)
   U02_DUST_EXTRAC_2_SWTCHD_OFF_I AT %M1216.6 : Bool;   // UNIT 02 DUST EXTRACCION 2 SWITCHED OFF INPUT
   U02_DUST_EXTRAC_2_SWTCH_ON_Q AT %M1216.7 : Bool;   // UNIT 02 DUST EXTRACCION 2 SWITCH ON OUTPUT
   U02_DUST_EXTRAC_2_SWTCH_OFF_Q AT %M1217.0 : Bool;   // UNIT 02 DUST EXTRACCION 2 SWITCH OFF OUTPUT
   "/////_UNIT_02_DUST_EXTRACTION_3_/////" AT %M1217.1 : Bool;   // /////_UNIT_02_DUST_EXTRACTION_3/////
   U02_DUST_EXTRAC_3_SWTCHD_ON_I AT %M1217.2 : Bool;   // UNIT 02 DUST EXTRACCION 3 SWITCHED ON INPUT (Flow Present)
   U02_DUST_EXTRAC_3_SWTCHD_OFF_I AT %M1217.3 : Bool;   // UNIT 02 DUST EXTRACCION 3 SWITCHED OFF INPUT
   U02_DUST_EXTRAC_3_SWTCH_OFF_Q AT %M1217.5 : Bool;   // UNIT 02 DUST EXTRACCION 3 SWITCH OFF OUTPUT
   "/////_UNIT_02_DUST_EXTRACTION_4_/////" AT %M1217.6 : Bool;   // /////_UNIT_02_DUST_EXTRACTION_4/////
   U02_DUST_EXTRAC_4_SWTCHD_ON_I AT %M1217.7 : Bool;   // UNIT 02 DUST EXTRACCION 4 SWITCHED ON INPUT (Flow Present)
   U02_DUST_EXTRAC_4_SWTCHD_OFF_I AT %M1218.0 : Bool;   // UNIT 02 DUST EXTRACCION 4 SWITCHED OFF INPUT
   U02_DUST_EXTRAC_4_SWTCH_OFF_Q AT %M1218.2 : Bool;   // UNIT 02 DUST EXTRACCION 4 SWITCH OFF OUTPUT
   "/////_UNIT_02_ANGULAR_LOCATOR_/////" AT %M1219.5 : Bool;
   U02_ANGULAR_LOCATOR_LCTD_I AT %I1578.0 : Bool;
   U02_ANGULAR_LOCATOR_RTND_I AT %I1578.1 : Bool;
   "/////_UNIT_02_AXIAL_LOCATOR_/////" AT %M1220.2 : Bool;
   U02_AXIAL_LOCATOR_LCTD_I AT %I1578.2 : Bool;
   U02_AXIAL_LOCATOR_RTND_I AT %I1578.3 : Bool;
   "/////_UNIT_02_STATION_4_BRUSH/////" AT %M1220.7 : Bool;   // /////_UNIT_02_STATION_4_BRUSH/////
   U02_ST4_BRUSH_LCTD_I AT %M1221.0 : Bool;   // UNIT 02 STATION 4 BRUSH LOCATED INPUT
   U02_ST4_BRUSH_RTND_I AT %M1221.1 : Bool;   // UNIT 02 STATION 4 BRUSH RETURNED INPUT
   U02_ST4_BRUSH_LCT_Q AT %Q1075.6 : Bool;   // UNIT 02 STATION 4 BRUSH LOCATE OUTPUT
   U02_ST4_BRUSH_RTN_Q AT %Q1075.7 : Bool;   // UNIT 02 STATION 4 BRUSH RETURN OUTPUT
   U01_HAT_UP_DOWN AT %I480.7 : Bool;   // UNIT 01 STATION 1 HAT UP / HAT DOWN
   U02_HAT_UP_DOWN AT %I1480.7 : Bool;   // UNIT 02 HAT UP / HAT DOWN
   U02_STA_1_PART_PRESENT AT %I1480.6 : Bool;   // UNIT 02 STATION 1 PART PRESENT
   U01_DUST_EXTRAC_4_SWTCH_ON_Q AT %Q66.0 : Bool;   // UNIT 01 DUST EXTRACCION 4 SWITCH ON OUTPUT
   U01_DUST_EXTRAC_1_SWTCH_ON_Q AT %Q66.2 : Bool;   // UNIT 01 DUST EXTRACCION 1 SWITCH ON OUTPUT
   KF76_SAFE_VALVE_ON AT %Q72.0 : Bool;   // KF76 SAFETY VALVE ON
   U01_DUST_EXTRAC_3_SWTCH_ON_Q AT %Q66.6 : Bool;   // UNIT 01 DUST EXTRACCION 3 SWITCH ON OUTPUT
   U02_DUST_EXTRAC_1_SWTCH_ON_Q AT %Q1066.2 : Bool;   // UNIT 02 DUST EXTRACCION 1 SWITCH ON OUTPUT
   U01_STA_1_PART_PRESENT_NC AT %I481.6 : Bool;   // UNIT 01 STATION 1 PART PRESENT NC
   U01_STA_1_PART_PRESENT_NO AT %I480.6 : Bool;   // UNIT 01 STATION 1 PART PRESENT NO
   U02_DUST_EXTRAC_4_SWTCH_ON_Q AT %Q1066.0 : Bool;   // UNIT 02 DUST EXTRACCION 4 SWITCH ON OUTPUT
   U02_DUST_EXTRAC_3_SWTCH_ON_Q AT %Q1067.0 : Bool;   // UNIT 02 DUST EXTRACCION 3 SWITCH ON OUTPUT
   DOWN_SEALING_U01_CLOSE_Q AT %Q72.1 : Bool;   // DOWN SEALING UNIT 01 STRUCTURE CLOSE OUTPUT
   DOWN_SEALING_U02_CLOSE_Q AT %Q1072.1 : Bool;   // DOWN SEALING UNIT 02 STRUCTURE CLOSE OUTPUT
   UP_SEALING_U02_OPEN_Q AT %Q1072.3 : Bool;   // UP SEALING UNIT 02 STRUCTURE CLOSE OUTPUT
   U02_ANGULAR_LOCATOR_RTN_Q AT %Q1074.0 : Bool;   // UNIT 01 ANGULAR LOCATOR RETURN OUTPUT
   DOWN_SEALING_U02_OPEN_Q AT %Q1072.2 : Bool;   // DOWN SEALING UNIT 02 STRUCTURE OPEN OUTPUT
   U02_ANGULAR_LOCATOR_LCT_Q AT %Q1073.7 : Bool;   // UNIT 01 ANGULAR LOCATOR LOCATE OUTPUT
   SAFETY_BRAKE_AXIS_Z23_UNBLCK_Q AT %Q1072.5 : Bool;   // SAFETY BRAKE AXIS Z23 UNBLOCK OUTPUT
   U01_AXIAL_LOCATOR_LCT_Q AT %Q74.1 : Bool;   // UNIT 01 AXIAL LOCATOR LOCATE OUTPUT
   UP_SEALING_U01_CLOSE_Q AT %Q72.4 : Bool;   // UP SEALING UNIT 01 STRUCTURE CLOSE (MOVE DOWN) OUTPUT
   U01_AXIAL_LOCATOR_RTN_Q AT %Q74.2 : Bool;   // UNIT 01 AXIAL LOCATOR RETURN OUTPUT
   U02_AXIAL_LOCATOR_LCT_Q AT %Q1074.1 : Bool;   // UNIT 01 AXIAL LOCATOR LOCATE OUTPUT
   UP_SEALING_U01_OPEN_Q AT %Q72.3 : Bool;   // UP SEALING UNIT 01 STRUCTURE OPEN (MOVE UP) OUTPUT
   UP_SEALING_U02_CLOSE_Q AT %Q1072.4 : Bool;   // UP SEALING UNIT 02 STRUCTURE OPEN OUTPUT
   DOWN_SEALING_U01_OPEN_Q AT %Q72.2 : Bool;   // DOWN SEALING UNIT 01 STRUCTURE OPEN OUTPUT
   SAFETY_BRAKE_AXIS_Z13_UNBLCK_Q AT %Q72.5 : Bool;   // SAFETY BRAKE AXIS Z13 UNBLOCK OUTPUT
   U02_AXIAL_LOCATOR_RTN_Q AT %Q1074.2 : Bool;   // UNIT 01 AXIAL LOCATOR RETURN OUTPUT
   U01_ANGULAR_LOCATOR_RTN_Q AT %Q74.0 : Bool;   // UNIT 01 ANGULAR LOCATOR RETURN OUTPUT
   U01_ANGULAR_LOCATOR_LCT_Q AT %Q73.7 : Bool;   // UNIT 01 ANGULAR LOCATOR LOCATE OUTPUT
END_VAR

VAR_GLOBAL   // PLC tag table "TAGS_IO_FIXTURES_UNIT_01"
   "/////_UNIT_01_FIXTURES_/////" AT %M2000.0 : Bool;   // /////_UNIT_01_FIXTURES_/////
   "/////_FIXTURE_1_UNIT_01_/////" AT %M2000.6 : Bool;   // /////_FIXTURE_1_UNIT_01_/////
   UNIT_01_FIX_1_GRIPPER_CLOSED_I AT %I60.4 : Bool;   // UNIT 01 FIXTURE 1 GRIPPER CLOSED INPUT
   UNIT_01_FIX_1_GRIPPER_OPEN_I AT %I60.5 : Bool;   // UNIT 01 FIXTURE 1 GRIPPER OPEN INPUT
   UNIT_01_FIX_1_CLOSE_GRIPPER_O AT %Q65.0 : Bool;   // UNIT 01 FIXTURE 1 GRIPPER CLOSE OUTPUT
   UNIT_01_FIX_1_OPEN_GRIPPER_O AT %Q65.1 : Bool;   // UNIT 01 FIXTURE 1 GRIPPER OPEN OUTPUT
   "/////_FIXTURE_2_UNIT_01_/////" AT %M2000.1 : Bool;   // /////_FIXTURE_2_UNIT_01_/////
   UNIT_01_FIX_2_GRIPPER_CLOSED_I AT %I60.6 : Bool;   // UNIT 01 FIXTURE 2 GRIPPER CLOSED INPUT
   UNIT_01_FIX_2_GRIPPER_OPEN_I AT %I60.7 : Bool;   // UNIT 01 FIXTURE 2 GRIPPER OPEN INPUT
   UNIT_01_FIX_2_CLOSE_GRIPPER_O AT %Q65.2 : Bool;   // UNIT 01 FIXTURE 2 GRIPPER CLOSE OUTPUT
   UNIT_01_FIX_2_OPEN_GRIPPER_O AT %Q65.3 : Bool;   // UNIT 01 FIXTURE 2 GRIPPER OPEN OUTPUT
   "/////_FIXTURE_3_UNIT_01_/////" AT %M2001.3 : Bool;   // /////_FIXTURE_3_UNIT_01_/////
   UNIT_01_FIX_3_GRIPPER_CLOSED_I AT %I61.0 : Bool;   // UNIT 01 FIXTURE 3 GRIPPER CLOSED INPUT
   UNIT_01_FIX_3_GRIPPER_OPEN_I AT %I61.1 : Bool;   // UNIT 01 FIXTURE 3 GRIPPER OPEN INPUT
   UNIT_01_FIX_3_CLOSE_GRIPPER_O AT %Q65.4 : Bool;   // UNIT 01 FIXTURE 3 GRIPPER CLOSE OUTPUT
   UNIT_01_FIX_3_OPEN_GRIPPER_O AT %Q65.5 : Bool;   // UNIT 01 FIXTURE 3 GRIPPER OPEN OUTPUT
   "/////_FIXTURE_4_UNIT_01_/////" AT %M2002.0 : Bool;   // /////_FIXTURE_4_UNIT_01_/////
   UNIT_01_FIX_4_GRIPPER_CLOSED_I AT %I61.2 : Bool;   // UNIT 01 FIXTURE 4 GRIPPER CLOSED INPUT
   UNIT_01_FIX_4_GRIPPER_OPEN_I AT %I61.3 : Bool;   // UNIT 01 FIXTURE 4 GRIPPER OPEN INPUT
   UNIT_01_FIX_4_CLOSE_GRIPPER_O AT %Q65.6 : Bool;   // UNIT 01 FIXTURE 4 GRIPPER CLOSE OUTPUT
   UNIT_01_FIX_4_OPEN_GRIPPER_O AT %Q65.7 : Bool;   // UNIT 01 FIXTURE 4 GRIPPER OPEN OUTPUT
END_VAR

VAR_GLOBAL   // PLC tag table "TAGS_IO_FIXTURES_UNIT_02"
   "/////_UNIT_02_FIXTURES_/////" AT %M4000.0 : Bool;   // /////_UNIT_02_FIXTURES_/////
   "/////_FIXTURE_1_UNIT_02_/////" AT %M4000.1 : Bool;   // /////_FIXTURE_1_UNIT_02_/////
   UNIT_02_FIX_1_GRIPPER_CLOSED_I AT %I1060.4 : Bool;   // UNIT 02 FIXTURE 1 GRIPPER CLOSED INPUT
   UNIT_02_FIX_1_GRIPPER_OPEN_I AT %I1060.5 : Bool;   // UNIT 02 FIXTURE 1 GRIPPER OPEN INPUT
   UNIT_02_FIX_1_CLOSE_GRIPPER_O AT %Q1065.0 : Bool;   // UNIT 02 FIXTURE 1 GRIPPER CLOSE OUTPUT
   UNIT_02_FIX_1_OPEN_GRIPPER_O AT %Q1065.1 : Bool;   // UNIT 02 FIXTURE 1 GRIPPER OPEN OUTPUT
   "/////_FIXTURE_2_UNIT_02_/////" AT %M4000.6 : Bool;   // /////_FIXTURE_2_UNIT_02_/////
   UNIT_02_FIX_2_GRIPPER_CLOSED_I AT %I1060.6 : Bool;   // UNIT 02 FIXTURE 2 GRIPPER CLOSED INPUT
   UNIT_02_FIX_2_GRIPPER_OPEN_I AT %I1060.7 : Bool;   // UNIT 02 FIXTURE 2 GRIPPER OPEN INPUT
   UNIT_02_FIX_2_CLOSE_GRIPPER_O AT %Q1065.2 : Bool;   // UNIT 02 FIXTURE 2 GRIPPER CLOSE OUTPUT
   UNIT_02_FIX_2_OPEN_GRIPPER_O AT %Q1065.3 : Bool;   // UNIT 02 FIXTURE 2 GRIPPER OPEN OUTPUT
   "/////_FIXTURE_3_UNIT_02_/////" AT %M4001.3 : Bool;   // /////_FIXTURE_3_UNIT_02_/////
   UNIT_02_FIX_3_GRIPPER_CLOSED_I AT %I1061.0 : Bool;   // UNIT 02 FIXTURE 3 GRIPPER CLOSED INPUT
   UNIT_02_FIX_3_GRIPPER_OPEN_I AT %I1061.1 : Bool;   // UNIT 02 FIXTURE 3 GRIPPER OPEN INPUT
   UNIT_02_FIX_3_CLOSE_GRIPPER_O AT %Q1065.4 : Bool;   // UNIT 02 FIXTURE 3 GRIPPER CLOSE OUTPUT
   UNIT_02_FIX_3_OPEN_GRIPPER_O AT %Q1065.5 : Bool;   // UNIT 02 FIXTURE 3 GRIPPER OPEN OUTPUT
   "/////_FIXTURE_4_UNIT_02_/////" AT %M4002.0 : Bool;   // /////_FIXTURE_4_UNIT_02_/////
   UNIT_02_FIX_4_GRIPPER_CLOSED_I AT %I1061.2 : Bool;   // UNIT 02 FIXTURE 4 GRIPPER CLOSED INPUT
   UNIT_02_FIX_4_GRIPPER_OPEN_I AT %I1061.3 : Bool;   // UNIT 02 FIXTURE 4 GRIPPER OPEN INPUT
   UNIT_02_FIX_4_CLOSE_GRIPPER_O AT %Q1065.6 : Bool;   // UNIT 02 FIXTURE 4 GRIPPER CLOSE OUTPUT
   UNIT_02_FIX_4_OPEN_GRIPPER_O AT %Q1065.7 : Bool;   // UNIT 02 FIXTURE 4 GRIPPER OPEN OUTPUT
END_VAR

VAR_GLOBAL   // PLC tag table "TAGS_IO_FIXTURES_UNIT_03"
   "/////MEASURING_UNIT/////" AT %M4500.0 : Bool;
   UMEAS_PUSHER_LCT_Q AT %M4500.1 : Bool;   // MEASURING UNIT LOCATE PUSHER OUTPUT
   UMEAS_PUSHER_RTN_Q AT %M4500.2 : Bool;   // MEASURING UNIT RETURN PUSHER OUTPUT
   UMEAS_PUSHER_UNLOCK_Q AT %M4500.3 : Bool;   // MEASURING UNIT UNLOCK PUSHER OUTPUT
   UMEAS_UNCLAMPED_I AT %M4500.4 : Bool;   // MEASURING UNIT PART UNCLAMPED INPUT
   UMEAS_CLAMPED_I AT %M4500.5 : Bool;   // MEASURING UNIT PART CLAMPED INPUT
   UMEAS_SPIN_CTRL_I AT %M4500.6 : Bool;   // MEASURING UNIT SPIN CONTROL INPUT
   UMEAS_PART_PRESENT_I AT %M4500.7 : Bool;   // MEASURING UNIT PART PRESENT INPUT
END_VAR

VAR_GLOBAL   // PLC tag table "TAGS_IO_OTHER_CLADDING"
   "/////_UNIT_01_STATION_3_PYROMETER_/////" AT %M1300.0 : Bool;   // /////_UNIT_01_STATION_3_PYROMETER/////
   "/////_UNIT_01_PART_PRESENT_CONTROL_/////" AT %M1300.2 : Bool;   // /////_UNIT_01_PART_PRESENT_CONTROL/////
   "/////_UNIT_01_JAW_CHUCK_GRIPPER_CONTROL/////" AT %M1300.4 : Bool;   // /////_UNIT_01_JAW_CHUCK_GRIPPER_CONTROL/////
   "/////_U01_PT100_TEMPERATURE_SENSORS_/////" AT %M1300.6 : Bool;   // /////_U01_PT100_TEMPERATURE_SENSORS_*/////
   U01_KF730_SENSOR_1 AT %MW1301 : Int;   // UNIT 01 KF730 SENSOR 1
   U01_KF730_SENSOR_2 AT %MW1303 : Int;   // UNIT 01 KF730 SENSOR 2
   U01_KF730_SENSOR_3 AT %MW1305 : Int;   // UNIT 01 KF730 SENSOR 3
   U01_KF730_SENSOR_4 AT %MW1307 : Int;   // UNIT 01 KF730 SENSOR 4
   U01_KF730_SENSOR_5 AT %MW1309 : Int;   // UNIT 01 KF730 SENSOR 5
   U01_KF730_SENSOR_6 AT %MW1311 : Int;   // UNIT 01 KF730 SENSOR 6
   U01_PT100_400_SENSOR_1 AT %MW1313 : Int;   // UNIT 01 PT100 400 SENSOR 1
   U01_PT100_400_SENSOR_2 AT %MW1315 : Int;   // UNIT 01 PT100 400 SENSOR 2
   U01_PT100_400_SENSOR_3 AT %MW1317 : Int;   // UNIT 01 PT100 400 SENSOR 3
   U01_PT100_400_SENSOR_4 AT %MW1319 : Int;   // UNIT 01 PT100 400 SENSOR 4
   U01_PT100_ENVIROMENT_1 AT %MW1321 : Int;   // UNIT 01 ENVIROMENT PT100 1
   U01_PT100_ENVIROMENT_2 AT %MW1323 : Int;   // UNIT 01 ENVIROMENT PT100 2
   U01_IN_POSITION AT %I500.6 : Bool;   // U01 READY TO MOVE. BOLT OK
   U01_TURN_CONTROL_FIXT AT %IW518 : Word;   // UNIT 01 FIXTURE TURNING CONTROL
   U01_AXIS_X13_ADVANCED_POS AT %I570.0 : Bool;   // AXIS X13 ADVANCED POSITION INPUT
   U01_AXIS_X13_GARAGE_POS AT %I570.1 : Bool;   // AXIS X13 GARAGE POSITION INPUT
   U01_AXIS_X13_RETURNED_POS AT %I570.2 : Bool;   // AXIS X13 RETURNED POSITION INPUT
   U01_AXIS_Z13_DOWN_POS AT %I570.3 : Bool;   // AXIS Z13 DOWN POSITION INPUT
   U01_AXIS_Z13_UP_POS AT %I570.4 : Bool;   // AXIS Z13 UP POSITION INPUT
   U01_AXIS_Z13_GARAGE_POS AT %I570.7 : Bool;   // AXIS Z13 GARAGE POSITION INPUT
   U01_STA_3_PRESSURE AT %IW526 : Word;   // UNIT 01 STATION 3 PRESSURE
   U01_LASER_COOLING_NOZZLE_FLOW_SP AT %I70.1 : Bool;   // UNIT 01 LASER COOLING NOZZLE FLOW SENSOR SETPOINT
   U01_LASER_COOLING_NOZZLE_TEMP_SP AT %I71.1 : Bool;   // UNIT 01 LASER COOLING NOZZLE TEMPERATURE SENSOR SETPOINT
   U01_LASER_COOLING_HEAD_FLOW_SP AT %I70.2 : Bool;   // UNIT 01 LASER COOLING HEAD FLOW SENSOR SETPOINT
   U01_LASER_COOLING_HEAD_TEMP_SP AT %I71.2 : Bool;   // UNIT 01 LASER COOLING HEAD TEMPERATURE SENSOR SETPOINT
   U01_LASER_COOLING_OUTPUT_FLOW_VALUE AT %MW1335 : Int;   // UNIT 01 LASER COOLING OUTPUT FLOW SENSOR VALUE
   U01_LASER_COOLING_OUTPUT_TEMP_VALUE AT %MW1337 : Word;   // UNIT 01 LASER COOLING OUTPUT TEMPERATURE SENSOR VALUE
   U01_LASER_COOLING_OUTPUT_FLOW_SP AT %I70.0 : Bool;   // UNIT 01 LASER COOLING OUTPUT FLOW SENSOR SETPOINT
   U01_LASER_COOLING_OUTPUT_TEMP_SP AT %I71.0 : Bool;   // UNIT 01 LASER COOLING OUTPUT TEMPERATURE SENSOR SETPOINT
   "/////_UNIT_02_STATION_3_PYROMETER/////" AT %M1338.0 : Bool;   // /////_UNIT_02_STATION_3_PYROMETER/////
   "/////_UNIT_02_PART_PRESENT_CONTROL/////" AT %M1338.2 : Bool;   // /////_UNIT_02_PART_PRESENT_CONTROL/////
   "/////_UNIT_02_JAW_CHUCK_GRIPPER_CONTROL/////" AT %M1338.4 : Bool;   // /////_UNIT_02_JAW_CHUCK_GRIPPER_CONTROL/////
   "/////_U02_PT100_TEMPERATURE_SENSORS_/////" AT %M1338.6 : Bool;   // /////_U02_PT100_TEMPERATURE_SENSORS_*/////
   U02_KF730_SENSOR_1 AT %MW1339 : Int;   // UNIT 02 KF730 SENSOR 1
   U02_KF730_SENSOR_2 AT %MW1341 : Int;   // UNIT 02 KF730 SENSOR 2
   U02_KF730_SENSOR_3 AT %MW1343 : Int;   // UNIT 02 KF730 SENSOR 3
   U02_KF730_SENSOR_4 AT %MW1345 : Int;   // UNIT 02 KF730 SENSOR 4
   U02_KF730_SENSOR_5 AT %MW1347 : Int;   // UNIT 02 KF730 SENSOR 5
   U02_KF730_SENSOR_6 AT %MW1349 : Int;   // UNIT 02 KF730 SENSOR 6
   U02_PT100_400_SENSOR_1 AT %MW1351 : Int;   // UNIT 02 PT100 400 SENSOR 1
   U02_PT100_400_SENSOR_2 AT %MW1353 : Int;   // UNIT 02 PT100 400 SENSOR 2
   U02_PT100_400_SENSOR_3 AT %MW1355 : Int;   // UNIT 02 PT100 400 SENSOR 3
   U02_PT100_400_SENSOR_4 AT %MW1357 : Int;   // UNIT 02 PT100 400 SENSOR 4
   U02_PT100_ENVIROMENT_1 AT %MW1359 : Int;   // UNIT 02 ENVIROMENT PT100 1
   U02_PT100_ENVIROMENT_2 AT %MW1361 : Int;   // UNIT 02 ENVIROMENT PT100 2
   "/////_UNIT_02_OTHERS_/////" AT %M1363.0 : Bool;   // /////_UNIT_02_OTHERS_/////
   U02_IN_POSITION AT %I1500.6 : Bool;   // U02 READY TO MOVE. BOLT OK
   U02_TURN_CONTROL_FIXT AT %IW1518 : Word;   // UNIT 01 FIXTURE TURNING CONTROL
   U02_X23_ADVANCED_POS AT %I1570.0 : Bool;   // AXIS X23 ADVANCED POSITION INPUT
   U02_X23_GARAGE_POS AT %I1570.1 : Bool;   // AXIS X23 GARAGE POSITION INPUT
   U02_X23_RETURNED_POS AT %I1570.2 : Bool;   // AXIS X23 RETURNED POSITION INPUT
   U02_Z23_DOWN_POS AT %I1570.3 : Bool;   // AXIS Z23 DOWN POSITION INPUT
   U02_Z23_UP_POS AT %I1570.4 : Bool;   // AXIS Z23 UP POSITION INPUT
   U02_Z23_GARAGE_POS AT %I1570.7 : Bool;   // AXIS Z23 GARAGE POSITION INPUT
   U02_LASER_COOLING_NOZZLE_FLOW_SP AT %I1070.1 : Bool;   // UNIT 01 LASER COOLING NOZZLE FLOW SENSOR SETPOINT
   U01_STA_1_PUSHER_W11_RTND AT %I470.1 : Bool;   // UNIT 01 PUSHER RETURNED
   U01_FIX_GRIPPER_CONTROL AT %IW468 : Word;   // UNIT 01 FIXTURE GRIPPER/JAW CHUCK CONTROL
   U02_FIX_GRIPPER_CONTROL AT %IW1468 : Word;   // UNIT 02 FIXTURE GRIPPER/JAW CHUCK CONTROL
   U02_STA_1_PUSHER_W21_RTND AT %I1470.1 : Bool;   // UNIT 02 PUSHER RETURNED
   "/////_UNIT_01_OTHERS_/////" AT %M1325.0 : Bool;   // /////_UNIT_01_OTHERS_/////
   U02_LASER_COOLING_NOZZLE_TEMP_VALUE AT %IW1652 : Int;   // UNIT 02 LASER COOLING NOZZLE TEMP VALUE
   U01_LASER_COOLING_NOZZLE_FLOW_VALUE AT %IW650 : Int;   // UNIT 01 LASER COOLING NOZZLE FLOW VALUE
   U02_LASER_COOLING_HEAD_TEMP_VALUE AT %ID1664 : DInt;   // UNIT 02 LASER COOLING HEAD TEMP VALUE
   U01_LASER_COOLING_HEAD_TEMP_VALUE AT %ID664 : DInt;   // UNIT 01 LASER COOLING HEAD TEMPERATURE VALUE
   U02_LASER_COOLING_NOZZLE_FLOW_VALUE AT %IW1650 : Int;   // UNIT 02 LASER COOLING NOZZLE FLOW VALUE
   U01_LASER_COOLING_NOZZLE_TEMP_VALUE AT %IW652 : Int;   // UNIT 01 LASER COOLING NOZZLE TEMPERATURE VALUE
   U02_LASER_COOLING_HEAD_FLOW_VALUE AT %ID1658 : DInt;   // UNIT 02 LASER COOLING HEAD FLOW VALUE
   U01_LASER_COOLING_HEAD_FLOW_VALUE AT %ID658 : DInt;   // UNIT 01 LASER COOLING HEAD FLOW VALUE
   U02_STA3_CLEANING_VALVE AT %Q68.0 : Bool;
   U01_STA3_CLEANING_VALVE AT %Q1068.0 : Bool;
   U01_TURCK_LD_PART_Q AT %Q606.3 : Bool;   // UNIT 01 BIMANUAL LOADED PART OUTPUT
   U01_TURCK_UNLD_PART_Q AT %Q606.1 : Bool;   // UNIT 01 BIMANUAL UNLOADED PART OUTPUT
   U01_TURCK_RESET_FAULTS_I AT %I606.4 : Bool;   // UNIT 01 BIMANUAL RESET FAULTS INPUT
   U01_TURCK_START_CYCLE_Q AT %Q606.7 : Bool;   // UNIT 01 BIMANUAL START CYCLE OUTPUT
   U01_TURCK_UNLD_PART_I AT %I606.0 : Bool;   // UNIT 01 BIMANUAL UNLOAD PART INPUT
   U01_TURCK_RESET_FAULTS_Q AT %Q606.5 : Bool;   // UNIT 01 BIMANUAL RESET FAULTS OUTPUT
   U01_TURCK_LD_PART_I AT %I606.2 : Bool;   // UNIT 01 BIMANUAL LOAD PART INPUT
   U01_TURCK_START_CYCLE_I AT %I606.6 : Bool;   // UNIT 01 BIMANUAL START CYCLE INPUT
   U01_PYRO_CURRENT_TRANSMISSION AT %ID3644 : Real;   // UNIT 01 PYROMETER CURRENT TRANSMISSION
   U01_PYRO_HEAD_TEMPERATURE AT %ID3608 : Real;   // UNIT 01 PYROMETER HEAD TEMPERATURE
   U02_PYRO_CURRENT_TRANSMISSION AT %ID3744 : Real;   // UNIT 02 PYROMETER CURRENT TRANSMISSION
   U02_PYRO_HEAD_TEMPERATURE AT %ID3708 : Real;   // UNIT 02 PYROMETER HEAD TEMPERATURE
   U01_PYRO_PROCESS_TEMPERATURE AT %ID3604 : Real;   // UNIT 01 PYROMETER PROCESS TEMPERATURE
   U01_PYRO_T2_TEMPERATURE AT %ID3632 : Real;   // UNIT 01 PYROMETER T2 TEMPERATURE
   U02_PYRO_PROCESS_TEMPERATURE AT %ID3704 : Real;   // UNIT 02 PYROMETER PROCESS TEMPERATURE
   U02_PYRO_CURRENT_EMISSIVITY AT %ID3740 : Real;   // UNIT 02 PYROMETER CURRENT EMISSIVITY
   U01_PYRO_CURRENT_EMISSIVITY AT %ID3640 : Real;   // UNIT 01 PYROMETER CURRENT EMISSIVITY
   U01_PYRO_T1_TEMPERATURE AT %ID3628 : Real;   // UNIT 01 PYROMETER T1 TEMPERATURE
   U01_PYRO_DEVICE_STATUS AT %ID3600 : Real;   // UNIT 01 PYROMETER DEVICE STATUS
   U02_PYRO_DEVICE_STATUS AT %ID3700 : Real;   // UNIT 02 PYROMETER DEVICE STATUS
   U02_PYRO_T1_TEMPERATURE AT %ID3728 : Real;   // UNIT 02 PYROMETER T1 TEMPERATURE
   U02_PYRO_T2_TEMPERATURE AT %ID3732 : Real;   // UNIT 02 PYROMETER T2 TEMPERATURE
   U02_LASER_COOLING_HEAD_TEMP_SP AT %I1071.2 : Bool;   // UNIT 02 LASER COOLING HEAD TEMPERATURE SENSOR SETPOINT
   U02_LASER_COOLING_NOZZLE_TEMP_SP AT %I1071.1 : Bool;   // UNIT 02 LASER COOLING NOZZLE TEMPERATURE SENSOR SETPOINT
   U02_LASER_COOLING_OUTPUT_FLOW_VALUE AT %MW1374 : Int;   // UNIT 02 LASER COOLING OUTPUT FLOW SENSOR VALUE
   U02_LASER_COOLING_HEAD_FLOW_SP AT %I1070.2 : Bool;   // UNIT 02 LASER COOLING HEAD FLOW SENSOR SETPOINT
   U02_LASER_COOLING_OUTPUT_FLOW_SP AT %I1070.0 : Bool;   // UNIT 02 LASER COOLING OUTPUT FLOW SENSOR SETPOINT
   U02_LASER_COOLING_OUTPUT_TEMP_VALUE AT %MW1376 : Word;   // UNIT 02 LASER COOLING OUTPUT TEMPERATURE SENSOR VALUE
   U02_LASER_COOLING_OUTPUT_TEMP_SP AT %I1071.0 : Bool;   // UNIT 02 LASER COOLING OUTPUT TEMPERATURE SENSOR SETPOINT
   U01_KF320_400_PT100_1 AT %IW512 : Int;   // UNIT 01 KF320 400ºC PT100 SENSOR 1
   U02_KF1320_400_PT100_2 AT %IW1516 : Int;   // UNIT 02 KF1320 400ºC PT100 SENSOR 2
   U01_KF320_400_PT100_2 AT %IW516 : Int;   // UNIT 01 KF320 400ºC PT100 SENSOR 2
   U02_KF1320_400_PT100_1 AT %IW1512 : Int;   // UNIT 02 KF1320 400ºC PT100 SENSOR 1
   U01_SHIELD_COOLING_FLOW_VALUE AT %IW690 : Int;   // UNIT 01 SHIELD COOLING FLOW VALUE
   U02_SHIELD_COOLING_TEMP_VALUE AT %IW1692 : Int;   // UNIT 02 SHIELD COOLING TEMPERATURE VALUE
   U01_SHIELD_COOLING_TEMP_VALUE AT %IW692 : Int;   // UNIT 01 SHIELD COOLING TEMPERATURE VALUE
   U02_SHIELD_COOLING_FLOW_VALUE AT %IW1690 : Int;   // UNIT 02 SHIELD COOLING FLOW VALUE
   U02_STA_3_PRESSURE AT %IW1526 : Word;   // UNIT 02 STATION 3 PRESSURE
END_VAR

VAR_GLOBAL   // PLC tag table "TAGS_IO_PROFINET_CLADDING"
   "/////_POWER_METER_/////" AT %M7000.0 : Bool;   // ///// POWER METER /////
   POWER_METER_TOTAL_APPARENT_FACTOR AT %MD7058 : Real;   // POWER METER TOTAL APPARENT FACTOR
   POWDER_METER_MAX_TOTAL_APPARENT_POWER AT %ID3560 : Real;   // POWDER METER MAX TOTAL APPARENT POWER
   POWER_FACTOR_L3 AT %ID3524 : Real;   // POWER FACTOR L3
   POWER_METER_ACTIVE_POWER_L3 AT %MD7046 : Real;   // POWER METER ACTIVE POWER L3
   POWER_METER_TOTAL_APPARENT_POWER AT %ID3532 : Real;   // POWER METEER TOTAL APPARENT POWER
   POWER_METER_ACTIVE_ENERGY_IMPORT_TARIFF_F AT %ID3536 : Real;   // POWER METER ACTIVE ENERGY IMPORT TARIFF (F)
   POWER_FACTOR_L1 AT %ID3516 : Real;   // POWER FACTOR L1
   POWER_METER_TOTAL_REACTIVE_POWER AT %ID3512 : Real;   // POWER METER TOTAL REACTIVE POWER
   POWER_METER_CURRENT_L3 AT %ID3556 : Real;   // POWER METER CURRENT L3
   POWER_METER_ACTIVE_ENERGY_IMPORT AT %MD7050 : Real;   // POWER METER ACTIVE ENERGY IMPORT TARRIF
   POWDER_METER_UNIVERSAL_COUNTER_1 AT %ID3544 : Real;   // POWDER METER UNIVERSAL COUNTER 1
   POWER_METER_ACTIVE_POWER_L1 AT %MD7038 : Real;   // POWER METER ACTIVE POWER L1
   POWER_METER_ACTIVE_POWER_L2 AT %MD7042 : Real;   // POWER METER ACTIVE POWER L2
   POWER_METER_ACTIVE_ENERGY_EXPORT_TARIFF_F AT %ID3540 : Real;   // POWER METER ACTIVE ENERGY EXPORT TARIFF (F)
   POWER_METER_TOTAL_ACTIVE_POWER AT %ID3528 : Real;   // POWER METER TOTAL ACTIVE POWER
   POWER_METER_CURRENT_L2 AT %ID3552 : Real;   // POWER METER CURRENT L2
   POWER_METER_CURRENT_L1 AT %ID3548 : Real;   // POWER METER CURRENT L1
   POWER_FACTOR_L2 AT %ID3520 : Real;   // POWER FACTOR L2
   POWER_METER_VOLTAGE_L2_L3 AT %ID3576 : Real;   // POWER METER VOLTAGE L2-L3
   POWER_METER_VOLTAGE_L2_N AT %ID3588 : Real;   // POWER METER VOLTAGE L2 N
   POWER_METER_VOLTAGE_L3_N AT %ID3592 : Real;   // POWER METER VOLTAGE L3 N
   POWER_METER_VOLTAGE_L1_N AT %ID3584 : Real;   // POWER METER VOLTAGE L1 N
   POWER_METER_LINE_FRECUENCY AT %ID3568 : Real;   // POWER METER LINE FRECUENCY
   POWER_METER_VOLTAGE_L3_L1 AT %ID3580 : Real;   // POWER METER VOLTAGE L3-L1
   POWER_METER_VOLTAGE_L1_L2 AT %ID3572 : Real;   // POWER METER VOLTAGE L1-L2
   POWER_METER_TOTAL_POWER_FACTOR AT %ID3564 : Real;   // POWER METER TOTAL POWER FACTOR
END_VAR

VAR_GLOBAL   // PLC tag table "TAGS_SAFETY_AXES"
   X23_SAFETY_IN AT %I6732.0 : "AXIS_SAFETY_IN";   // CLADDING NCU AXIS 3
   E20_SAFETY_OUT AT %Q6892.0 : "AXIS_SAFETY_OUT";   // CLADDING NX X104 AXIS 13
   C14_SAFETY_IN AT %I6844.0 : "AXIS_SAFETY_IN";   // CLADDING NX X105 AXIS 10
   C14_SAFETY_OUT AT %Q6844.0 : "AXIS_SAFETY_OUT";   // CLADDING NX X105 AXIS 10
   C23_SAFETY_OUT AT %Q6924.0 : "AXIS_SAFETY_OUT";   // CLADDING NX X104 AXIS 15
   UNIT_3_AXES AT %M6796.3 : Bool;
   C22_SAFETY_OUT AT %Q6956.0 : "AXIS_SAFETY_OUT";   // CLADDING NX X104 AXIS 17
   C24_SAFETY_IN AT %I6940.0 : "AXIS_SAFETY_IN";   // CLADDING NX X103 AXIS 16
   C23_SAFETY_IN AT %I6924.0 : "AXIS_SAFETY_IN";   // CLADDING NX X104 AXIS 15
   C12_SAFETY_OUT AT %Q6860.0 : "AXIS_SAFETY_OUT";   // CLADDING NX X105 AXIS 11
   Z11_SAFETY_OUT AT %Q6988.0 : "AXIS_SAFETY_OUT";   // CLADDING NX X102 AXIS 19
   C12_SAFETY_IN AT %I6860.0 : "AXIS_SAFETY_IN";   // CLADDING NX X105 AXIS 11
   Z13_SAFETY_IN AT %I6716.0 : "AXIS_SAFETY_IN";   // CLADDING NCU AXIS 2
   Z13_SAFETY_OUT AT %Q6716.0 : "AXIS_SAFETY_OUT";   // CLADDING NCU AXIS 2
   C13_SAFETY_OUT AT %Q6828.0 : "AXIS_SAFETY_OUT";   // CLADDING NX X105 AXIS 9
   C11_SAFETY_OUT AT %Q6812.0 : "AXIS_SAFETY_OUT";   // CLADDING NX X105 AXIS 8
   C21_SAFETY_OUT AT %Q6908.0 : "AXIS_SAFETY_OUT";   // CLADDING NX X104 AXIS 14
   X13_SAFETY_IN AT %I6700.0 : "AXIS_SAFETY_IN";   // CLADDING NCU AXIS 1
   Z21_SAFETY_IN AT %I7004.0 : "AXIS_SAFETY_IN";   // CLADDING NX X102 AXIS 20
   E10_SAFETY_IN AT %I6796.0 : "AXIS_SAFETY_IN";   // CLADDING NX X105 AXIS 7
   Z21_SAFETY_OUT AT %Q7004.0 : "AXIS_SAFETY_OUT";   // CLADDING NX X102 AXIS 20
   Z23_SAFETY_OUT AT %Q6748.0 : "AXIS_SAFETY_OUT";   // CLADDING NCU AXIS 4
   C24_SAFETY_OUT AT %Q6940.0 : "AXIS_SAFETY_OUT";   // CLADDING NX X103 AXIS 16
   Z11_SAFETY_IN AT %I6988.0 : "AXIS_SAFETY_IN";   // CLADDING NX X102 AXIS 19
   X23_SAFETY_OUT AT %Q6732.0 : "AXIS_SAFETY_OUT";   // CLADDING NCU AXIS 3
   Z23_SAFETY_IN AT %I6748.0 : "AXIS_SAFETY_IN";   // CLADDING NCU AXIS 4
   C11_SAFETY_IN AT %I6812.0 : "AXIS_SAFETY_IN";   // CLADDING NX X105 AXIS 8
   C21_SAFETY_IN AT %I6908.0 : "AXIS_SAFETY_IN";   // CLADDING NX X104 AXIS 14
   C31_SAFETY_OUT AT %Q7020.0 : "AXIS_SAFETY_OUT";   // CLADDING NX X103 AXIS 23
   E10_SAFETY_OUT AT %Q6796.0 : "AXIS_SAFETY_OUT";   // CLADDING NX X105 AXIS 7
   UNIT_2_AXES AT %M6796.2 : Bool;
   C13_SAFETY_IN AT %I6828.0 : "AXIS_SAFETY_IN";   // CLADDING NX X105 AXIS 9
   C31_SAFETY_IN AT %I7020.0 : "AXIS_SAFETY_IN";   // CLADDING NX X103 AXIS 23
   E20_SAFETY_IN AT %I6892.0 : "AXIS_SAFETY_IN";   // CLADDING NX X104 AXIS 13
   UNIT_1_AXES AT %M6796.1 : Bool;
   C22_SAFETY_IN AT %I6956.0 : "AXIS_SAFETY_IN";   // CLADDING NX X104 AXIS 17
   X13_SAFETY_OUT AT %Q6700.0 : "AXIS_SAFETY_OUT";   // CLADDING NCU AXIS 1
END_VAR

TYPE "UDT_Feeder Line"
// stored: IsFailsafeCompliant false
   STRUCT
      GAS_FLOW_RATE_ACTUAL : Real;   // GAS FLOW RATE - ACTUAL
      GAS_FLOW_RATE_AUTO : Real;   // GAS FLOW RATE - AUTO
      GAS_FLOW_RATE_MANUAL : Real;   // GAS FLOW RATE - MANUAL
      DISC_SPEED_ACTUAL : Real;   // DISC SPEED - ACTUAL
      DISC_SPEED_AUTO : Real;   // DISC SPEED - AUTO
      DISC_SPEED_MANUAL : Real;   // DISC SPEED - MANUAL
      STIRRER_SPEED_ACTUAL : Real;   // STIRRER SPEED - ACTUAL
      STIRRER_SPEED_AUTO : Real;   // STIRRER SPEED - AUTO
      STIRRER_SPEED_MANUAL : Real;   // STIRRER SPEED - MANUAL
      HOPPER_TEMP_ACTUAL : Real;   // HOPPER TEMP - ACTUAL
      HOPPER_TEMP_AUTO : Real;   // HOPPER TEMP - AUTO
      HOPPER_TEMP_MANUAL : Real;   // HOPPER TEMP - MANUAL
      HEATER_ON_MANUAL_REQUEST : Bool;   // HEATER ON MANUAL REQUEST
      HEATER_OFF_MANUAL_REQUEST : Bool;   // HEATER OFF MANUAL REQUEST
      HEATER_STATUS : Byte;   // HEATER STATUS
      HOPPER_ON_MANUAL_REQUEST : Bool;   // HOPPER ON MANUAL REQUEST
      HOPPER_OFF_MANUAL_REQUEST : Bool;   // HOPPER OFF MANUAL REQUEST
      HOPPER_STATUS : Byte;   // HOPPER STATUS
      START_SEQUENCE_GAS_STEPS : Int;   // START SEQUENCE GAS STEPS
      START_SEQUENCE_DISK_STEPS : Int;   // START SEQUENCE DISK STEPS
      STOP_SEQUENCE_GAS_STEPS : Int;   // STOP SEQUENCE GAS STEPS
      STOP_SEQUENCE_DISK_STEPS : Int;   // STOP SEQUENCE DISK STEPS
      STOP_SEQUENCE_PAUSE_STEP : Int;   // STOP SEQUENCE PAUSE STEP
      DISC_SPEED_WARNING_UPPER_LIMIT : Real;   // DISC SPEED - WARNING UPPER LIMIT
      DISC_SPEED_ALARM_UPPER_LIMIT : Real;   // DISC SPEED - ALARM UPPER LIMIT
      DISC_SPEED_WARNING_LOWER_LIMIT : Real;   // DISC SPEED - WARNING LOWER LIMIT
      DISC_SPEED_ALARM_LOWER_LIMIT : Real;   // DISC SPEED - ALARM LOWER LIMIT
      GAS_FLOW_RATE_WARNING_UPPER_LIMIT : Real;   // GAS FLOW RATE - WARNING UPPER LIMIT
      GAS_FLOW_RATE_ALARM_UPPER_LIMIT : Real;   // GAS FLOW RATE - ALARM UPPER LIMIT
      GAS_FLOW_RATE_WARNING_LOWER_LIMIT : Real;   // GAS FLOW RATE - WARNING LOWER LIMIT
      GAS_FLOW_RATE_ALARM_LOWER_LIMIT : Real;   // GAS FLOW RATE - ALARM LOWER LIMIT
      STIRRER_SPEED_WARNING_UPPER_LIMIT : Real;   // STIRRER SPEED - WARNING UPPER LIMIT
      STIRRER_SPEED_ALARM_UPPER_LIMIT : Real;   // STIRRER SPEED - ALARM UPPER LIMIT
      STIRRER_SPEED_WARNING_LOWER_LIMIT : Real;   // STIRRER SPEED - WARNING LOWER LIMIT
      STIRRER_SPEED_ALARM_LOWER_LIMIT : Real;   // STIRRER SPEED - ALARM LOWER LIMIT
      HOPPER_TEMP_ALARM_UPPER_LIMIT : Real;   // HOPPER TEMP - ALARM UPPER LIMIT
      PRESSURE_VALUE_CURRENT_SENSOR : Real;   // PRESSURE VALUE - CURRENT SENSOR
   END_STRUCT;
END_TYPE

TYPE "UDT_Hopper Line"
// stored: IsFailsafeCompliant false
   STRUCT
      STIRRER_SPEED_ACTUAL : DInt;   // STIRRER SPEED - ACTUAL
      STIRRER_SPEED_MANUAL : DInt;   // STIRRER SPEED - MANUAL
      STIRRER_SPEED_AUTO : DInt;   // STIRRER SPEED - AUTO
      TEMP_UPPER_JACKET_ACTUAL : Real;   // TEMP UPPER JACKET - ACTUAL
      TEMP_UPPER_JACKET_MANUAL : Real;   // TEMP UPPER JACKET - MANUAL
      TEMP_UPPER_JACKET_AUTO : Real;   // TEMP UPPER JACKET - AUTO
      TEMP_LOWER_JACKET_ACTUAL : Real;   // TEMP LOWER JACKET - ACTUAL
      TEMP_LOWER_JACKET_MANUAL : Real;   // TEMP LOWER JACKET - MANUAL
      TEMP_LOWER_JACKET_AUTO : Real;   // TEMP LOWER JACKET - AUTO
      MAX_WEIGHT_ACTUAL : Real;   // MAX WEIGHT - ACTUAL
      MAX_WEIGHT_MANUAL : Real;   // MAX WEIGHT - MANUAL
      TOTAL_WEIGHT_ACTUAL : Real;   // TOTAL WEIGHT - ACTUAL
      HOPPER_WEIGHT_ACTUAL : Real;   // HOPPER WEIGHT - ACTUAL
      HOPPER_WEIGHT_MANUAL : Real;   // HOPPER WEIGHT - MANUAL
      POWDER_WEIGHT_ACTUAL : Real;   // POWDER WEIGHT - ACTUAL
      HOPPER_COVER_ACTUAL : Real;   // HOPPER COVER- ACTUAL
      HOPPER_COVER_MANUAL : Real;   // HOPPER COVER - MANUAL
      HOPPER_COVER_AUTO : Real;   // HOPPER COVER - AUTO
      FEEDING_COVER_ACTUAL : Real;   // FEEDING COVER - ACTUAL
      FEEDER_DISK_PRESSURE_ACTUAL : Real;   // FEEDER DISK PRESSURE- ACTUAL
      POWDER_FEEDER_WEIGHT_ACTUAL : Real;   // POWDER FEEDER WEIGHT ACTUAL
      TRANSFER_POWDER_SEQ_START : Bool;   // TRANSFER POWDER SEQ - START
      TRANSFER_POWDER_SEQ_STOP : Bool;   // TRANSFER POWDER SEQ - STOP
      PRESSURIZE_GAS_VALVE_START : Bool;   // PRESSURIZE GAS VALVE - START
      PRESSURIZE_GAS_VALVE_STOP : Bool;   // PRESSURIZE GAS VALVE - STOP
      RELIEVE_GAS_VALVE_START : Bool;   // RELIEVE GAS VALVE - START
      RELIEVE_GAS_VALVE_STOP : Bool;   // RELIEVE GAS VALVE - STOP
      CLEANING_AIR_VALVE_START : Bool;   // CLEANING AIR VALVE - START
      CLEANING_AIR_VALVE_STOP : Bool;   // CLEANING AIR VALVE - STOP
      LOAD_FEEDER_SEQUENCE_START : Bool;   // LOAD FEEDER SEQUENCE - START
      LOAD_FEEDER_SEQUENCE_STOP : Bool;   // LOAD FEEDER SEQUENCE - STOP
      STIRRER_STARTED : Bool;   // STIRRER - STARTED
      TEMP_UPPER_JACKET_STARTED : Bool;   // TEMP UPPER JACKET - STARTED
      TEMP_LOWER_JACKET_STARTED : Bool;   // TEMP LOWER JACKET - STARTED
      HOPPER_COVER_STARTED : Bool;   // HOPPER COVER - STARTED
   END_STRUCT;
END_TYPE

TYPE "UDT_Hopper_Actions"
// stored: IsFailsafeCompliant false
   STRUCT
      IKG_HOPPER_START : Bool;
      FEEDING_COVER_START : Bool;
      L1_HOPPER_LOW_START : Bool;
      L2_HOPPER_LOW_START : Bool;
      STIRRER_SPEED_START : Bool;
      VIBRATION_MOTOR_SPEED_START : Bool;
      TEMP_UPPER_JACKET_START : Bool;
      TEMP_LOWER_JACKET_START : Bool;
   END_STRUCT;
END_TYPE

TYPE "U03_MEAS_STATION_FACE_A.U03_FACE_A_MEAS_Method.Trigger calibration.Inputs"
// stored: IsFailsafeCompliant false
   STRUCT
      Force { ExternalAccessible := 'False'; ExternalVisible := 'False'; ExternalWritable := 'False'} : Bool;
   END_STRUCT;
END_TYPE

TYPE "U03_MEAS_STATION_FACE_B.U03_FACE_B_MEAS_Method.Trigger calibration.Inputs"
// stored: IsFailsafeCompliant false
   STRUCT
      Force { ExternalAccessible := 'False'; ExternalVisible := 'False'; ExternalWritable := 'False'} : Bool;
   END_STRUCT;
END_TYPE

TYPE "AUTO_SINGLE_SEMI_MANUAL"
// stored: IsFailsafeCompliant false
   STRUCT
      MANUAL_INPUT : Bool;   // MANUAL INPUT / MANUAL MODE INPUT
      SEMIAUTO_INPUT : Bool;   // SEMIAUTO INPUT / SEMIAUTOMATIC MODE INPUT
      AUTOMATIC_INPUT : Bool;   // AUTOMATIC INPUT / AUTOMATIC MODE INPUT
      SINGLE_INPUT : Bool;   // SINGLE CYCLE INPUT / SINGLE MODE INPUT
      NO_MODE_INPUT : Bool;   // NO MODE INPUT
      JOG_INPUT : Bool;   // JOG INPUT / JOG MODE INPUT
      TOOL_CHANGE_INPUT : Bool;   // TOOL CHANGE INPUT / TOOL CHANGE MODE INPUT
      CHANGE_GENERAL_CONDITIONS : Bool;   // CHANGE GENERAL CONDITIONS / CHANGE MODE GENERAL CONDITIONS
      CHANGE_INITIAL_CONDITIONS : Bool;   // CHANGE INITIAL CONDITIONS / CHANGE MODE INITIAL CONDITIONS
      MANUAL_REQUEST : Bool;   // MANUAL REQUEST / MANUAL MODE REQUEST
      SEMIAUTO_REQUEST : Bool;   // SEMIAUTO REQUEST / SEMIAUTOMATIC MODE REQUEST
      AUTOMATIC_REQUEST : Bool;   // AUTOMATIC REQUEST / AUTOMATIC MODE REQUEST
      SINGLE_REQUEST : Bool;   // SINGLE CYCLE REQUEST / SINGLE MODE REQUEST
      NO_MODE_REQUEST : Bool;   // NO MODE REQUEST
      NO_MODE_P_REQUEST_P : Bool;   // NO MODE REQUEST POSITIVE PULSE / NO MODE POSITIVE PULSE REQUEST
      NO_MODE_N_REQUEST_P : Bool;   // NO MODE REQUEST NEGATIVE PULSE / NO MODE NEGATIVE PULSE REQUEST
      JOG_REQUEST : Bool;   // JOG REQUEST / JOG MODE REQUEST
      TOOL_CHANGE_REQUEST : Bool;   // TOOL CHANGE REQUEST / TOOL CHANGE MODE REQUEST
      CHANGE_TO_MANUAL : Bool;   // CHANGE TO MANUAL MODE
      CHANGE_TO_MANUAL_P : Bool;   // CHANGE TO MANUAL PULSE / CHANGE TO MANUAL MODE PULSE
      CHANGE_TO_SEMIAUTO : Bool;   // CHANGE TO SEMIAUTO MODE / CHANGE TO SEMIAUTOMATIC MODE
      CHANGE_TO_AUTOMATIC : Bool;   // CHANGE TO AUTOMATIC MODE
      CHANGE_TO_SINGLE : Bool;   // CHANGE TO SINGLE CYCLE MODE / CHANGE TO SINGLE MODE
      CHANGE_TO_NO_MODE : Bool;   // CHANGE TO NO MODE
      CHANGE_TO_JOG_MODE : Bool;   // CHANGE TO JOG MODE
      CHANGE_TO_TOOL_CHG_MODE : Bool;   // CHANGE TO TOOL CHANGE MODE
      CHANGE_MODE_SEQ_RUN : Bool;   // CHANGE MODE SEQUENCE RUNNING
      MANUAL_SELECTED : Bool;   // MANUAL MODE SELECTED
      SEMIAUTO_SELECTED : Bool;   // SEMIAUTO MODE SELECTED / SEMIAUTOMATIC MODE SELECTED
      AUTOMATIC_SELECTED : Bool;   // AUTOMATIC MODE SELECTED
      SINGLE_SELECTED : Bool;   // SINGLE CYCLE MODE SELECTED / SINGLE MODE SELECTED
      NO_MODE_SELECTED : Bool;   // NO MODE MODE SELECTED / NO MODE SELECTED
      JOG_SELECTED : Bool;   // JOG MODE SELECTED
      TOOL_CHANGE_MODE_SELECTED : Bool;   // TOOL CHANGE MODE SELECTED
      AUTO_SINGLE_SEMI_SELECTED : Bool;   // AUTO / SEMIAUTO / SINGLE CYCLE MODE SELECTED / AUTO SINGLE SEMI MODE SELECTED
      MANUAL_SELECTED_MEMORY : Bool;   // MEMORY CHANGE MANUAL MODE / MANUAL MODE SELECTED MEMORY
      SEMI_SELECTED_MEMORY : Bool;   // MEMORY CHANGE MANUAL MODE / SEMI MODE SELECTED MEMORY
      AUTO_SELECTED_MEMORY : Bool;   // MEMORY CHANGE MANUAL MODE / AUTO MODE SELECTED MEMORY
      SINGLE_SELECTED_MEMORY : Bool;   // MEMORY CHANGE MANUAL MODE / SINGLE MODE SELECTED MEMORY
      JOG_SELECTED_MEMORY : Bool;   // MEMORY CHANGE JOG MODE / JOG MODE SELECTED MEMORY
      CHANGE_GENERAL_CONDITIONS_HELP : Bool;   // MODE CHANGE FAULT / CHANGE MODE GENERAL CONDITIONS HELP
      CHANGE_TO_MANUAL_ALARM : Bool;   // MANUAL MODE CHANGE FAULT / CHANGE TO MANUAL MODE ALARM
      CHANGE_TO_SEMIAUTO_ALARM : Bool;   // SEMIAUTO MODE CHANGE FAULT / CHANGE TO SEMIAUTO MODE ALARM
      CHANGE_TO_AUTO_ALARM : Bool;   // AUTOMATIC MODE CHANGE FAULT / CHANGE TO AUTO MODE ALARM
      CHANGE_TO_SINGLE_ALARM : Bool;   // SINGLE CYCLE MODE CHANGE FAULT / CHANGE TO SINGLE MODE ALARM
      CHANGE_TO_NO_MODE_ALARM : Bool;   // NO MODE CHANGE FAULT / CHANGE TO NO MODE ALARM
      CHANGE_TO_JOG_MODE_ALARM : Bool;   // JOG MODE CHANGE FAULT / CHANGE TO JOG MODE ALARM
      ELECTRONIC_HANDWEHELL_ACTIVE : Bool;   // ELECTRONIC HANDWEHELL ACTIVE
      OPTIONS : Struct
         SGM : Bool;   // SGM MACHINE
         GM : Bool;   // GM MACHINE
         FORD : Bool;   // FORD MACHINE
         ETXETAR : Bool;   // ETXETAR MACHINE
      END_STRUCT;
   END_STRUCT;
END_TYPE

TYPE "CYCLES"
// stored: IsFailsafeCompliant false
   STRUCT
      GENERAL_CONDITIONS : Bool;   // CHANGE GENERAL CONDITIONS / CHANGE CYCLE GENERAL CONDITIONS
      INITIAL_CONDITIONS : Bool;   // CHANGE INITIAL CONDITIONS / CHANGE CYCLE INITIAL CONDITIONS
      ENABLE_REQUEST : Bool;   // ENABLE REQUEST
      DISABLE_REQUEST : Bool;   // DISABLE REQUEST
      TOGGLE_COMMAND_P : Bool;   // TOGGLE COMAND PULSE / TOGGLE COMMAND PULSE
      WARNING_GONE : Bool;   // TOGGLE COMMAND AUXILIARY / WARNING GONE
      GENERAL_CONDITIONS_HELP : Bool;   // GENERAL CONDITIONS HELP / CHANGE CYCLE GENERAL CONDITIONS HELP
      INITIAL_CONDITIONS_HELP : Bool;   // INITIAL CONDITIONS HELP / CHANGE CYCLE INITIAL CONDITIONS HELP
      CYCLE_SELECTED : Bool;   // MODE SELECTED / CYCLE SELECTED
      CYCLE_SELECTED_AUX : Bool;   // AUXILIARY MODE SELECTED / CYCLE SELECTED AUXILIARY
      CYCLE_COMPLETED : Bool;   // COMPLETED / CYCLE COMPLETED
      MACHINE_EMPTY : Bool;   // MACHINE EMPTY
      MACHINE_EMPTY_MANUAL_LOAD_SELECTED : Bool;   // MACHINE EMPTY WITH MANUAL LOAD SELECTED / MACHINE EMPTY MANUAL LOAD SELECTED
      MACHINE_EMPTY_WO_MANUAL_LOAD_SELECTED : Bool;   // MACHINE EMPTY WITHOUT MANUAL LOAD SELECTED
      RESET_FULL_DEPTH_DRY_CYCLE_DISABLED : Bool;   // RESET DEPTHS WHEN DRY CYCLE DISABLED / RESET FULL DEPTH DRY CYCLE DISABLED
      RESET_FULL_DEPTHS_AUX : Bool;   // RESET FULL DEPTHS AUXILIARY
      CYCLE_SEOC : Bool;   // CYCLE STOP END OF CYCLE
      CYCLE_IS : Bool;   // CYCLE IMMEDIATE STOP
   END_STRUCT;
END_TYPE

TYPE "MODES"
// stored: IsFailsafeCompliant false
   STRUCT
      GENERAL_CONDITIONS : Bool;   // CHANGE GENERAL CONDITIONS / GENERAL CONDITIONS
      INITIAL_CONDITIONS : Bool;   // CHANGE INITIAL CONDITIONS / INITIAL CONDITIONS
      ENABLE_REQUEST : Bool;   // ENABLE REQUEST
      DISABLE_REQUEST : Bool;   // DISABLE REQUEST
      TOGGLE_COMMAND_P : Bool;   // TOGGLE COMAND PULSE / TOGGLE COMMAND PULSE
      TOGGLE_COMMAND : Bool;   // TOGGLE COMMAND AUXILIARY / TOGGLE COMMAND
      GENERAL_CONDITIONS_HELP : Bool;   // GENERAL CONDITIONS HELP
      INITIAL_CONDITIONS_HELP : Bool;   // INITIAL CONDITIONS HELP
      MODE_SELECTED : Bool;   // MODE SELECTED
      WARNING_GONE : Bool;   // WARNING GONE
   END_STRUCT;
END_TYPE

TYPE "DIAGNOSTIC_MOD"
// stored: IsFailsafeCompliant false
   STRUCT
      CHANNEL_1_STATE : Bool;   // CHANNEL 1 STATE
      CHANNEL_2_STATE : Bool;   // CHANNEL 2 STATE
      CHANNEL_3_STATE : Bool;   // CHANNEL 3 STATE
      CHANNEL_4_STATE : Bool;   // CHANNEL 4 STATE
      CHANNEL_1_ALARM : Bool;   // CHANNEL 1 ALARM
      CHANNEL_2_ALARM : Bool;   // CHANNEL 2 ALARM
      CHANNEL_3_ALARM : Bool;   // CHANNEL 3 ALARM
      CHANNEL_4_ALARM : Bool;   // CHANNEL 4 ALARM
      MOD_ERROR_ALARM : Bool;   // MOD ERROR ALARM
   END_STRUCT;
END_TYPE

TYPE "HT10_ENABLE_CHANGE"
// stored: IsFailsafeCompliant false
   STRUCT
      GENERAL_CONDITIONS : Bool;   // GENERAL CONDITIONS
      INTIAL_CONDITIONS : Bool;   // INTIAL CONDITIONS
      MANUAL_REQUEST : Bool;   // MANUAL REQUEST
      GLOBAL_REQUEST : Bool;   // GLOBAL REQUEST
      GLOBAL_REQUEST_RETURN : Bool;   // GLOBAL REQUEST RETURN
      CONTROL_PANEL : Bool;   // CONTROL PANEL
      SELECTED : Bool;   // SELECTED
      HELP : Bool;   // HELP
      PULSE : Bool;   // PULSE
      PULSE_1 : Bool;   // PULSE 1
      PULSE_2 : Bool;   // PULSE 2
      PULSE_3 : Bool;   // PULSE 3
      PULSE_4 : Bool;   // PULSE 4
      GENERAL_CONDITIONS_HELP : Bool;   // GENERAL CONDITIONS HELP
      INITIAL_CONDITIONS_HELP : Bool;   // INITIAL CONDITIONS HELP
   END_STRUCT;
END_TYPE

TYPE "HT10_INPUTS"
// stored: IsFailsafeCompliant false
   STRUCT
      SPARE_0_0 : Bool;   // SPARE 0 0
      RESET_FAULT_I : Bool;   // HT10 RESET FAULT INPUT
      SPARE_0_2 : Bool;   // SPARE 0 2
      SPARE_0_3 : Bool;   // SPARE 0 3
      SPARE_0_4 : Bool;   // SPARE 0 4
      SPARE_0_5 : Bool;   // SPARE 0 5
      SPARE_0_6 : Bool;   // SPARE 0 6
      SPARE_0_7 : Bool;   // SPARE 0 7
      SPARE_1_0 : Bool;   // SPARE 1 0
      SPARE_1_1 : Bool;   // SPARE 1 1
      U1 : Bool;   // SELECT MANUAL MODE
      U2 : Bool;   // SELECT REFERENCE MODE
      SPARE_1_4 : Bool;   // SPARE 1 4
      U3 : Bool;   // SELECT SEMIAUTO MODE
      U4 : Bool;   // SPARE 1 6
      U_OPTION_I : Bool;   // HT10 U OPTION INPUT
      SPARE_2 : Byte;   // SPARE 2
      SPARE_3_0 : Bool;   // SPARE 3 0
      SPARE_3_1 : Bool;   // SPARE 3 1
      SPARE_3_2 : Bool;   // SPARE 3 2
      SPARE_3_3 : Bool;   // SPARE 3 3
      SPARE_3_4 : Bool;   // SPARE 3 4
      SPARE_3_5 : Bool;   // SPARE 3 5
      JOG_MIINUS_I : Bool;   // HT10 JOG MIINUS INPUT
      JOG_PLUS_I : Bool;   // HT10 JOG PLUS INPUT
      U16 : Bool;   // SPARE 3 0
      U15 : Bool;   // SPARE 3 1
      U14 : Bool;   // SPARE 3 2
      U13 : Bool;   // SPARE 3 3
      U12 : Bool;   // SPARE 3 4
      U11 : Bool;   // SPARE 3 5
      U10 : Bool;   // SPARE 3 5
      U9 : Bool;   // SPARE 3 5
      RAPID_I : Bool;   // HT10 RAPID INPUT
      SPARE_5_1 : Bool;   // SPARE 5 1
      SPARE_5_2 : Bool;   // SPARE 5 2
      U5 : Bool;   // SPARE 5 3
      U6 : Bool;   // SPARE 5 4
      U7 : Bool;   // SPARE 5 5
      U8 : Bool;   // SPARE 5 6
      SPARE_5_7 : Bool;   // SPARE 5 7
      NC_STOP_I : Bool;   // HT10 NC STOP INPUT
      NC_START_I : Bool;   // HT10 NC START INPUT
      OVERRIDE_I : Byte;   // HT10 OVERRIDE INPUT
   END_STRUCT;
END_TYPE

TYPE "HT10_OUTPUTS"
// stored: IsFailsafeCompliant false
   STRUCT
      SPARE_0_0 : Bool;   // SPARE 0 0
      RESET_FAULT_Q : Bool;   // HT10 RESET FAULT OUTPUT
      SPARE_1 : Byte;   // SPARE 1
      SPARE_2_0 : Bool;   // SPARE 2 0
      SPARE_2_1 : Bool;   // SPARE 2 1
      SPARE_2_2 : Bool;   // SPARE 2 2
      SPARE_2_3 : Bool;   // SPARE 2 3
      SPARE_2_4 : Bool;   // SPARE 2 4
      SPARE_2_5 : Bool;   // SPARE 2 5
      SPARE_2_6 : Bool;   // SPARE 2 6
      JOG_PLUS_Q : Bool;   // HT10 JOG PLUS OUTPUT
      SPARE_3_0 : Bool;   // SPARE 3 0
      SPARE_3_1 : Bool;   // SPARE 3 1
      SPARE_3_2 : Bool;   // SPARE 3 2
      SPARE_3_3 : Bool;   // SPARE 3 3
      SPARE_3_4 : Bool;   // SPARE 3 4
      SPARE_3_5 : Bool;   // SPARE 3 5
      JOG_MIINUS_Q : Bool;   // HT10 JOG MIINUS OUTPUT
      SPARE_3_7 : Bool;   // SPARE 3 7
      SPARE_4 : Byte;   // SPARE 4
      RAPID_Q : Bool;   // HT10 RAPID OUTPUT
      SPARE_5_1 : Bool;   // SPARE 5 1
      SPARE_5_2 : Bool;   // SPARE 5 2
      SPARE_5_3 : Bool;   // SPARE 5 3
      SPARE_5_4 : Bool;   // SPARE 5 4
      SPARE_5_5 : Bool;   // SPARE 5 5
      SPARE_5_6 : Bool;   // SPARE 5 6
      SPARE_5_7 : Bool;   // SPARE 5 7
      NC_STOP_Q : Bool;   // HT10 NC STOP OUTPUT
      NC_START_Q : Bool;   // HT10 NC START OUTPUT
   END_STRUCT;
END_TYPE

TYPE "MPP_INPUTS"
// stored: IsFailsafeCompliant false
   STRUCT
      I_S59_E_STOP_OVERRIDE : Bool;   // S59 - S11 HAND HELD PANEL ENABLE / S59 - S11 EMERGENCY STOP OVERRIDE
      I_S60 : Bool;   // S60 - S11 BA MODE ENABLE / S60 - EXTENSION KEY
      I_S62_HG_CONNECTION : Bool;   // S62 - XS12:13 HG CONNECTION
      I_F21 : Bool;   // F21 FUNCTION KEY - RESET
      I_WS1_1 : Bool;   // F1 FUNCTION KEY - CONTINUOUS CYCLE // BA WS1/1 / WS1/1 - CONTINUOUS CYCLE
      I_WS1_2 : Bool;   // F6 FUNCTION KEY - ONE CYCLE // BA WS1/2 / WS1/2 - SINGLE CYCLE
      I_WS1_3 : Bool;   // F11 FUNCTION KEY - STEP BY STEP CYCLE // BA WS1/3 / WS1/3 - STEP BY STEP CYCLE
      I_WS1_4 : Bool;   // F16 FUNCTION KEY - SETUP // BA WS1/4 / WS1/4 - SETUP
      I_S1 : Bool;   // MPP483 KEY - CONTROL ON / S1 KEY - CONTROL ON
      I_S2 : Bool;   // MPP483 KEY - START / S2 KEY - START
      I_S3 : Bool;   // MPP483 KEY - HOME POSITION / S3 KEY - HOME POSITION
      I_S4 : Bool;   // MPP483 KEY - RESET FAULT / S4 KEY - RESET FAULT
      I_S51 : Bool;   // S51 EXTENSION KEY - / S51 - EXTENSION KEY
      I_S14 : Bool;   // S5 CUSTOMER KEY - / S14 - USER KEY
      I_WS4_KEY_POS_0 : Bool;   // MPP483 KEY - POSITION 0 / WS4 KEY - POSITION 0
      I_S15 : Bool;   // MPP483 KEY - / S15 KEY - USER KEY
      I_WS5_1_RAP_TRAV_OVERR : Bool;   // WS5/1 - RAPID TRAVERSE OVERRIDE
      I_WS5_2_RAP_TRAV_OVERR : Bool;   // WS5/2 - RAPID TRAVERSE OVERRIDE
      I_WS5_4_RAP_TRAV_OVERR : Bool;   // WS5/4 - RAPID TRAVERSE OVERRIDE
      I_WS5_8_RAP_TRAV_OVERR : Bool;   // WS5/8 - RAPID TRAVERSE OVERRIDE
      I_S61 : Bool;   // S61 - SR KEY / S61 - EXTENSION KEY
      I_WS4_KEY_POS_1 : Bool;   // WS4 KEY - POSITION 1
      I_WS4_KEY_POS_2 : Bool;   // WS4 KEY - POSITION 2
      I_WS4_KEY_POS_3 : Bool;   // WS4 KEY - POSITION 3
      I_S52 : Bool;   // S52 EXTENSION KEY - / S52 - EXTENSION KEY
      I_S7 : Bool;   // MPP483 KEY - CONTROL OFF / S7 KEY - CONTROL OFF
      I_S8 : Bool;   // MPP483 KEY - REQUEST STOP END OF CYCLE / S8 KEY - REQUEST STOP END OF CYCLE
      I_S9 : Bool;   // MPP483 KEY - IMMEDIATE STOP / S9 KEY - IMMEDIATE STOP
      I_S10 : Bool;   // MPP483 KEY - UNLOCK SAFETY DOORS / S10 KEY - UNLOCK SAFETY DOORS
      I_S13 : Bool;   // S11 - EMERGENCY STOP / S13 - EMERGENCY STOP
      I_S53 : Bool;   // S53 EXTENSION KEY - / S53 - EXTENSION KEY
      I_3_7 : Bool;   // NOT USED
      I_DT1 : Bool;   // DT1 - DIRECT CONTROL KEY / DT1 - DIRECT KEY
      I_DT2 : Bool;   // DT2 - DIRECT CONTROL KEY / DT2 - DIRECT KEY
      I_DT3 : Bool;   // DT3 - DIRECT CONTROL KEY / DT3 - DIRECT KEY
      I_DT4 : Bool;   // DT4 - DIRECT CONTROL KEY / DT4 - DIRECT KEY
      I_DT5 : Bool;   // DT5 - DIRECT CONTROL KEY / DT5 - DIRECT KEY
      I_DT6 : Bool;   // DT6 - DIRECT CONTROL KEY / DT6 - DIRECT KEY
      I_DT7 : Bool;   // DT7 - DIRECT CONTROL KEY / DT7 - DIRECT KEY
      I_DT8 : Bool;   // DT8 - DIRECT CONTROL KEY / DT8 - DIRECT KEY
      I_DT9 : Bool;   // DT9 - DIRECT CONTROL KEY / DT9 - DIRECT KEY
      I_DT10 : Bool;   // DT10 - DIRECT CONTROL KEY / DT10 - DIRECT KEY
      I_DT11 : Bool;   // DT11 - DIRECT CONTROL KEY / DT11 - DIRECT KEY
      I_DT12 : Bool;   // DT12 - DIRECT CONTROL KEY / DT12 - DIRECT KEY
      I_DT13 : Bool;   // DT13 - DIRECT CONTROL KEY / DT13 - DIRECT KEY
      I_DT14 : Bool;   // DT14 - DIRECT CONTROL KEY / DT14 - DIRECT KEY
      I_DT15 : Bool;   // DT15 - DIRECT CONTROL KEY / DT15 - DIRECT KEY
      I_DT16 : Bool;   // DT16 - DIRECT CONTROL KEY / DT16 - DIRECT KEY
      I_WS3_1_SPIND_OVERR : Bool;   // WS3/1 - SPINDLE OVERRIDE
      I_WS3_2_SPIND_OVERR : Bool;   // WS3/2 - SPINDLE OVERRIDE
      I_WS3_4_SPIND_OVERR : Bool;   // WS3/4 - SPINDLE OVERRIDE
      I_WS3_8_SPIND_OVERR : Bool;   // WS3/8 - SPINDLE OVERRIDE
      I_S57 : Bool;   // S57 EXTENSION KEY - / S57 - EXTENSION KEY
      I_S58 : Bool;   // S58 EXTENSION KEY - / S58 - EXTENSION KEY
      I_6_6 : Bool;   // NOT USED
      I_6_7 : Bool;   // NOT USED
      I_WS2_1_FEED_OVERR : Bool;   // WS2/1 - FEEDRATE OVERRIDE
      I_WS2_2_FEED_OVERR : Bool;   // WS2/2 - FEEDRATE OVERRIDE
      I_WS2_4_FEED_OVERR : Bool;   // WS2/4 - FEEDRATE OVERRIDE
      I_WS2_8_FEED_OVERR : Bool;   // WS2/8 - FEEDRATE OVERRIDE
      I_WS2_16_FEED_OVERR : Bool;   // WS2/16 - FEEDRATE OVERRIDE
      I_S54 : Bool;   // S54 EXTENSION KEY - / S54 - EXTENSION KEY
      I_S55 : Bool;   // S55 EXTENSION KEY - / S55 - EXTENSION KEY
      I_S56 : Bool;   // S56 EXTENSION KEY - / S56 - EXTENSION KEY
      I_F1 : Bool;   // F1 FUNCTION KEY - CONTINUOUS CYCLE
      I_F2 : Bool;   // F2 FUNCTION KEY - AUTOMATIC MODE
      I_F3 : Bool;   // F3 FUNCTION KEY - SINGLE BLOCK
      I_F4 : Bool;   // F4 FUNCTION KEY - NC STOP
      I_F5 : Bool;   // F5 FUNCTION KEY - NC START
      I_F6 : Bool;   // F6 FUNCTION KEY - ONE CYCLE / F6 FUNCTION KEY - SINGLE CYCLE
      I_F7 : Bool;   // F7 FUNCTION KEY - MDA MODE
      I_F8 : Bool;   // F8 FUNCTION KEY - NEXT AXES
      I_F9 : Bool;   // F9 FUNCTION KEY - FEEDRATE STOP
      I_F10 : Bool;   // F10 FUNCTION KEY - FEEDRATE START
      I_F11 : Bool;   // F11 FUNCTION KEY - STEP BY STEP CYCLE
      I_F12 : Bool;   // F12 FUNCTION KEY - JOG MODE
      I_F13 : Bool;   // F13 FUNCTION KEY - (X1 - W) AXES / F13 FUNCTION KEY - (X11 - W) AXES
      I_F14 : Bool;   // F14 FUNCTION KEY - (Y1 - E) AXES / F14 FUNCTION KEY - (Y11 - E) AXES
      I_F15 : Bool;   // F15 FUNCTION KEY - Z11 AXIS
      I_F16 : Bool;   // F16 FUNCTION KEY - SETUP MODE
      I_F17 : Bool;   // F17 FUNCTION KEY - REFERENCE POINT MODE
      I_F18 : Bool;   // F18 FUNCTION KEY - (A - U1 - C) AXES / F18 FUNCTION KEY - (A11 - U11 - C) AXES
      I_F19 : Bool;   // F18 FUNCTION KEY - B AXIS / F19 FUNCTION KEY - B AXIS
      I_F20 : Bool;   // F18 FUNCTION KEY - (Q1 - Z12) AXES / F20 FUNCTION KEY - (Q11 - Z12) AXES
      I_F22 : Bool;   // F22 FUNCTION KEY - INCREMENTAL MODE
      I_F23 : Bool;   // F23 FUNCTION KEY - MINUS DIRECTION
      I_F24 : Bool;   // F24 FUNCTION KEY - RAPID
      I_F25 : Bool;   // F25 FUNCTION KEY - PLUS DIRECTION
      I_BYTE_11 : Byte;   // RESERVED / RESERVE
      I_WS2_1_FEED_OVERRIDE : Bool;   // WS2/1 - FEEDRATE OVERRIDE
      I_WS2_2_FEED_OVERRIDE : Bool;   // WS2/2 - FEEDRATE OVERRIDE
      I_WS2_4_FEED_OVERRIDE : Bool;   // WS2/4 - FEEDRATE OVERRIDE
      I_WS2_8_FEED_OVERRIDE : Bool;   // WS2/8 - FEEDRATE OVERRIDE
      I_WS2_16_FEED_OVERRIDE : Bool;   // WS2/16 - FEEDRATE OVERRIDE
      I_12_5 : Bool;   // NOT USED
      I_12_6 : Bool;   // NOT USED
      I_12_7 : Bool;   // NOT USED
      I_WS3_1_SPIND_OVERRIDE : Bool;   // WS3/1 - SPINDLE OVERRIDE
      I_WS3_2_SPIND_OVERRIDE : Bool;   // WS3/2 - SPINDLE OVERRIDE
      I_WS3_4_SPIND_OVERRIDE : Bool;   // WS3/4 - SPINDLE OVERRIDE
      I_WS3_8_SPIND_OVERRIDE : Bool;   // WS3/8 - SPINDLE OVERRIDE
      I_WS3_16_SPIND_OVERRIDE : Bool;   // WS3/16 - SPINDLE OVERRIDE
      I_13_5 : Bool;   // NOT USED
      I_13_6 : Bool;   // NOT USED
      I_13_7 : Bool;   // NOT USED
      HANDWHEEL_1_COUNTER_READ : Int;   // HANDWHEEL 1 - COUNTER STATUS / HANDWHEEL 1 - COUNTER READING
      HANDWHEEL_2_COUNTER_READ : Int;   // HANDWHEEL 2 - COUNTER STATUS / HANDWHEEL 2 - COUNTER READING
   END_STRUCT;
END_TYPE

TYPE "MPP_OUTPUTS"
// stored: IsFailsafeCompliant false
   STRUCT
      O_HS1 : Bool;   // MPP483 LAMP - CONTROL ON / LAMP - CONTROL ON
      O_HS2 : Bool;   // MPP483 LAMP - START / LAMP - START
      O_HS3 : Bool;   // MPP483 LAMP - HOME / LAMP - HOME
      O_HS4 : Bool;   // MPP483 LAMP - RESET FAULT / LAMP - RESET FAULT
      O_HS14 : Bool;   // MPP483 LAMP - / LAMP -
      O_HS15 : Bool;   // MPP483 LAMP - / LAMP -
      O_HS7 : Bool;   // MPP483 LAMP - CONTROL OFF / LAMP - CONTROL OFF
      O_HS8 : Bool;   // MPP483 LAMP - STOP END OF CYCLE / LAMP - STOP END OF CYCLE
      O_HS9 : Bool;   // MPP483 LAMP - IMMEDIATE STOP / LAMP - IMMEDIATE STOP
      O_HS10 : Bool;   // MPP483 LAMP - SAFETY DOOR CLOSED & LOCKED / LAMP - SAFETY DOOR CLOSED AND LOCKED
      O_1_2 : Bool;   // NOT USED
      O_1_3 : Bool;   // NOT USED
      O_1_4 : Bool;   // NOT USED
      O_1_5 : Bool;   // NOT USED
      O_1_6 : Bool;   // NOT USED
      O_1_7 : Bool;   // NOT USED
      O_H51 : Bool;   // H51 EXTENSION KEY - / H51 - EXTENSION KEY
      O_H52 : Bool;   // H52 EXTENSION KEY - / H52 - EXTENSION KEY
      O_H53 : Bool;   // H53 EXTENSION KEY - / H53 - EXTENSION KEY
      O_H54 : Bool;   // H54 EXTENSION KEY - / H54 - EXTENSION KEY
      O_H55 : Bool;   // H55 EXTENSION KEY - / H55 - EXTENSION KEY
      O_H56 : Bool;   // H56 EXTENSION KEY - / H56 - EXTENSION KEY
      O_H57 : Bool;   // H57 EXTENSION KEY - / H57 - EXTENSION KEY
      O_H58 : Bool;   // H58 EXTENSION KEY - / H58 - EXTENSION KEY
      O_H59 : Bool;   // H59 EXTENSION KEY - / H59 - EXTENSION KEY
      O_H60 : Bool;   // H60 EXTENSION KEY - / H60 - EXTENSION KEY
      O_HS13 : Bool;   // HS13 - FEEDBACK EMERGENCY STOP
      O_H61_SR_PUSH_BUTTON : Bool;   // H61 - SR KEY / H61 - SR PUSH BUTTON
      O_3_4 : Bool;   // NOT USED
      O_3_5 : Bool;   // NOT USED
      O_3_6 : Bool;   // NOT USED
      O_3_7 : Bool;   // NOT USED
      O_HF1 : Bool;   // MPP483 LAMP - CONTINUOUS CYCLE / LAMP - CONTINUOUS CYCLE
      O_HF2 : Bool;   // MPP483 LAMP - AUTOMATIC MODE / LAMP - AUTOMATIC MODE
      O_HF3 : Bool;   // MPP483 LAMP - SINGLE BLOCK / LAMP - SINGLE BLOCK
      O_HF4 : Bool;   // MPP483 LAMP - NC STOP / LAMP - NC STOP
      O_HF5 : Bool;   // MPP483 LAMP - NC START / LAMP - NC START
      O_HF6 : Bool;   // MPP483 LAMP - ONE CYCLE / LAMP - SINGLE CYCLE
      O_HF7 : Bool;   // MPP483 LAMP - MDA MODE / LAMP - MDA MODE
      O_HF8 : Bool;   // MPP483 LAMP - NEXT AXES / LAMP - NEXT AXES
      O_HF9 : Bool;   // MPP483 LAMP - FEEDRATE STOP / LAMP - FEEDRATE STOP
      O_HF10 : Bool;   // MPP483 LAMP - FEEDRATE START / LAMP - FEEDRATE START
      O_HF11 : Bool;   // MPP483 LAMP - STEP BY STEP CYCLE / LAMP - STEP BY STEP CYCLE
      O_HF12 : Bool;   // MPP483 LAMP - JOG MODE / LAMP - JOG MODE
      O_HF13 : Bool;   // MPP483 LAMP - (X1 - W) AXES / LAMP - (X1 - W) AXES
      O_HF14 : Bool;   // MPP483 LAMP - (Y1 - E) AXES / LAMP - (Y1 - E) AXES
      O_HF15 : Bool;   // MPP483 LAMP - Z11 AXIS / LAMP - Z11 AXIS
      O_HF16 : Bool;   // MPP483 LAMP - SETUP MODE / LAMP - SETUP MODE
      O_HF17 : Bool;   // MPP483 LAMP - REFERENCE POINT MODE / LAMP - REFERENCE POINT MODE
      O_HF18 : Bool;   // MPP483 LAMP - (A - U1 - C) AXES / LAMP - (A - U1 - C) AXES
      O_HF19 : Bool;   // MPP483 LAMP - B AXIS / LAMP - B AXIS
      O_HF20 : Bool;   // MPP483 LAMP - (Q1 - Z12) AXES / LAMP - (Q1 - Z12) AXES
      O_HF21 : Bool;   // MPP483 LAMP - RESET / LAMP - RESET
      O_HF22 : Bool;   // MPP483 LAMP - INCREMENTAL MODE / LAMP - INCREMENTAL MODE
      O_HF23 : Bool;   // MPP483 LAMP - MINUS DIRECTION / LAMP - MINUS DIRECTION
      O_HF24 : Bool;   // MPP483 LAMP - RAPID / LAMP - RAPID
      O_HF25 : Bool;   // MPP483 LAMP - PLUS DIRECTION / LAMP - PLUS DIRECTION
      O_7_1 : Bool;   // NOT USED
      O_7_2 : Bool;   // NOT USED
      O_7_3 : Bool;   // NOT USED
      O_7_4 : Bool;   // NOT USED
      O_7_5 : Bool;   // NOT USED
      O_7_6 : Bool;   // NOT USED
      O_7_7 : Bool;   // NOT USED
   END_STRUCT;
END_TYPE

TYPE "TEST_24HRS"
// stored: IsFailsafeCompliant false
   STRUCT
      Day : Byte;
      Month : Byte;
      Year : Byte;
      Hour : Byte;
      Minute : Byte;
      Second : Byte;
      mSecond : Byte;
      Spare : Int;
   END_STRUCT;
END_TYPE

TYPE "GLOBAL_DATA_CLADDING"
// stored: IsFailsafeCompliant false
   STRUCT
      NO_MACHINE_CYCLE_RUN_P : Bool;   // NO CYCLE MACHINE RUN PROGRAM / NO MACHINE CYCLE RUNNING PULSE
      ANY_MACHINE_CYCLE_RUN_P : Bool;   // ANY MACHINE CYCLE RUN PROGRAM / ANY MACHINE CYCLE RUNNING PULSE
      NO_MACHINE_CYCLE_RUN_HOPPER_UNIT_01_P : Bool;   // NO CYCLE MACHINE RUN PROGRAM / NO MACHINE CYCLE RUNNING HOPPER UNIT 01 PULSE
      ANY_HOPPER_UNIT_01_CYCLE_RUN_P : Bool;   // ANY MACHINE CYCLE RUN PROGRAM / ANY HOPPER UNIT 01 CYCLE RUNNING PULSE
      NO_MACHINE_CYCLE_RUN_HOPPER_UNIT_02_P : Bool;   // NO CYCLE MACHINE RUN PROGRAM / NO MACHINE CYCLE RUNNING HOPPER UNIT 02 PULSE
      ANY_HOPPER_UNIT_02_CYCLE_RUN_P : Bool;   // ANY MACHINE CYCLE RUN PROGRAM / ANY HOPPER UNIT 02 CYCLE RUNNING PULSE
      ANY_MACHINE_CYCLE_RUN : Bool;   // ANY MACHINE CYCLE RUN / ANY MACHINE CYCLE RUNNING
      ANY_UNIT_01_CYCLE_RUN : Bool;   // ANY MACHINE CYCLE RUN / ANY UNIT 01 CYCLE RUNNING
      ANY_UNIT_02_CYCLE_RUN : Bool;   // ANY MACHINE CYCLE RUN / ANY UNIT 02 CYCLE RUNNING
      ANY_HOPPER_UNIT_01_CYCLE_RUN : Bool;   // ANY MACHINE CYCLE RUN / ANY HOPPER UNIT 01 CYCLE RUNNING
      ANY_HOPPER_UNIT_02_CYCLE_RUN : Bool;   // ANY MACHINE CYCLE RUN / ANY HOPPER UNIT 02 CYCLE RUNNING
      ANY_HOPPER_1_UNIT_01_CYCLE_RUN : Bool;   // ANY HOPPER 1 UNIT 01 CYCLE RUNNING
      ANY_HOPPER_2_UNIT_01_CYCLE_RUN : Bool;   // ANY HOPPER 2 UNIT 01 CYCLE RUNNING
      ANY_HOPPER_1_UNIT_02_CYCLE_RUN : Bool;   // ANY HOPPER 1 UNIT 02 CYCLE RUNNING
      ANY_HOPPER_2_UNIT_02_CYCLE_RUN : Bool;   // ANY HOPPER 2 UNIT 02 CYCLE RUNNING
      ANY_HOPPER_3_UNIT_02_CYCLE_RUN : Bool;   // ANY HOPPER 3 UNIT 02 CYCLE RUNNING
      ANY_POWDER_FEEDER_RUN : Bool;   // ANY POWDER FEEDER RUNNING
      AUX0 : Bool;   // AUXILIARY 0
      AUX1 : Bool;   // AUXILIARY 1
      AUX2 : Bool;   // AUXILIARY 2
      AUX3 : Bool;   // AUXILIARY 3
      AUX4 : Bool;   // AUXILIARY 4
      AUX5 : Bool;   // AUXILIARY 5
      AUX6 : Bool;   // AUXILIARY 6
      AUX7 : Bool;   // AUXILIARY 7
      AUX8 : Bool;   // AUXILIARY 7
      AUX9 : Bool;   // AUXILIARY 7
      AUX10 : Bool;   // AUXILIARY 7
      AUX11 : Bool;   // AUXILIARY 7
   END_STRUCT;
END_TYPE

TYPE "WINCC_HMI_LINES"
// stored: IsFailsafeCompliant false
   STRUCT
      WINCC_LINE_REQUEST_RIGHT : Bool;   // RIGHT REQUEST
      WINCC_LINE_REQUEST_LEFT : Bool;   // LEFT REQUEST
      WINCC_LINE_CONDITIONS_RIGHT : Bool;   // RIGHT CONDITIONS
      WINCC_LINE_CONDITIONS_LEFT : Bool;   // LEFT CONDITIONS
      WINCC_LINE_ACTIVE_RIGHT : Bool;   // RIGHT ACTIVE
      WINCC_LINE_ACTIVE_LEFT : Bool;   // LEFT ACTIVE
      WINCC_LINE_STATUS_1_RIGHT : Bool;   // RIGHT STATUS 1
      WINCC_LINE_STATUS_1_LEFT : Bool;   // LEFT STATUS 1
      WINCC_LINE_STATUS_2_RIGHT : Bool;   // RIGHT STATUS 2
      WINCC_LINE_STATUS_2_LEFT : Bool;   // LEFT STATUS 2
      WINCC_LINE_STATUS_3_RIGHT : Bool;   // RIGHT STATUS 3
      WINCC_LINE_STATUS_3_LEFT : Bool;   // LEFT STATUS 3
      WINCC_LINE_STATUS_4_RIGHT : Bool;   // RIGHT STATUS 4
      WINCC_LINE_STATUS_4_LEFT : Bool;   // LEFT STATUS 4
      WINCC_LINE_STATUS_5_RIGHT : Bool;   // RIGHT STATUS 5
      WINCC_LINE_STATUS_5_LEFT : Bool;   // LEFT STATUS 5
   END_STRUCT;
END_TYPE

